// TwinCAT 3 PLC project PLC_TMO_VAC
// Title: PLC_TMO_VAC
// Company: SLAC - LCLS
// ProjectVersion: 0.0.0
// ProgramVersion: 3.1.4022.7
// CompilerDefines: K
// libraries:
//   LCLS General, * (SLAC)
//   LCLS Vacuum, * (SLAC - LCLS)
//   LCLSVacuumSerialDriverLib, * (SLAC - LCLS)
//   PMPS, * (SLAC - LCLS)
//   Tc2_SerialCom, * (Beckhoff Automation GmbH)
//   Tc2_Standard, * (Beckhoff Automation GmbH)
//   Tc2_System, * (Beckhoff Automation GmbH)
//   Tc3_Module, * (Beckhoff Automation GmbH)
// project tree:
//   / ComTask.TcTTO, FSVTask.TcTTO, PlcTask.TcTTO
//   DUTs/ E_STATES.TcDUT
//   GVLs/ GVL_COM.TcGVL, GVL_DREAM_ECAT.TcGVL, GVL_FEE_Device.TcGVL, GVL_FSV_PMPS.TcGVL, GVL_FS_Devices.TcGVL, GVL_Hutch_Gauges.TcGVL, GVL_Hutch_Pumps.TcGVL, GVL_Hutch_Valves.TcGVL, GVL_IP1_ECAT.TcGVL, GVL_PMPS.TcGVL, GVL_Variables.TcGVL
//   POUs/ DIAGNOSTICS.TcPOU, FB_VRC_NO_FFO_VLS.TcPOU, F_Turbo_Protection_ILK.TcPOU, MAIN.TcPOU, PRG_COM.TcPOU, PRG_FEE.TcPOU, PRG_FSV.TcPOU, PRG_FSV_Interfaces.TcPOU, PRG_Hutch_Beamline_Valves.TcPOU, PRG_Hutch_Gauges.TcPOU, PRG_Hutch_Ion_Pumps.TcPOU, PRG_HV_SAFETY.TcPOU, PRG_IP1_ECAT_Interfaces.TcPOU, PRG_PMPS.TcPOU, PRG_Roughing_Pumps.TcPOU, PRG_ECAT_COMM_CHECK.TcPOU
// real-time tasks:
//   TASK PlcTask: cycle T#10ms, priority 20, ADS port 350
//   TASK ComTask: cycle T#11ms, priority 30, ADS port 351
//   TASK FSVTask: cycle T#2ms, priority 15, ADS port 352
// I/O:
//   DEVICE Device 1 (EtherCAT), AmsNetId 172.21.132.78.2.1
//     B940-R20-CX0 (EK1200) [EK1200-5000 EtherCAT Power supply (2A E-Bus)]
//       CX0_E1 (EL2202) [EL2202 2Ch. Dig. Output 24V, 0.5A]
//       CX0_E1A (EL2202) [EL2202 2Ch. Dig. Output 24V, 0.5A]
//       Term 113 (EL2202) [EL2202 2Ch. Dig. Output 24V, 0.5A]
//       CX0_E2_EXILK (EL1008) [EL1008 8Ch. Dig. Input 24V, 3ms]
//       CX0_E5 (EL6070) [EL6070 1Ch. Licensing-Terminal]
//       CX0_E6_QPC1 (EL3064) [EL3064 4Ch. Ana. Input 0-10V]
//       CX0_E7_QPC1 (EL1004) [EL1004 4Ch. Dig. Input 24V, 3ms]
//       CX0_E8_QPC1 (EL2794) [EL2794 4Ch. Dig. Output 24V AC/DC, 2A, short-circuit-proof]
//       CX0_E9_QPC2 (EL3064) [EL3064 4Ch. Ana. Input 0-10V]
//       CX0_E10_QPC2 (EL1004) [EL1004 4Ch. Dig. Input 24V, 3ms]
//       CX0_E11_QPC2 (EL2794) [EL2794 4Ch. Dig. Output 24V AC/DC, 2A, short-circuit-proof]
//       CX0_E12 (EL6001) [EL6001 Interface (RS232)]
//       CX0_E13 (EK1122) [EK1122 2 port EtherCAT junction]
//         IP1_ECAT [EL6695 EtherCAT Bridge terminal (Secondary)]
//         DREAM_ECAT [EL6695 EtherCAT Bridge terminal (Secondary)]
//       PMPS_PRE [EL6692 EtherCAT Bridge terminal (Primary)]
//       CX0_EK1110 [EK1110 EtherCAT extension]
//     B940_R20_EK0 (EK1100) [EK1100 EtherCAT Coupler (2A E-Bus)]
//       R20_EK0_E1_MKS937B (EL3064)
//       R20_EK0_E2_MKS937B (EL3064) [EL3064 4Ch. Ana. Input 0-10V]
//       R20_EK0_E3_MKS937B (EL2794) [EL2794 4Ch. Dig. Output 24V AC/DC, 2A, short-circuit-proof]
//       R20_EK0_SIP (EL3174-0002) [EL3174-0002 4Ch. Ana. Input +/-10V, +/-20mA 16 Bit, Isolated Channels]
//       R20_EK0_E4_MKS937B (EL9505) [EL9505 Power supply terminal 5V]
//       R20_EK0_E5_MKS937B (EL1124)
//       R20_EK0_E5A_MKS937B (EL1124) [EL1124 4Ch. Dig. Input 5V, 10µs, Sensor Power]
//       R20_EK0_E6_MKS937B (EK1110) [EK1110 EtherCAT extension]
//     B940_K4S20_EK0  (EK1100) [EK1100 EtherCAT Coupler (2A E-Bus)]
//       K4S20-E1-FSV (EL1004)
//       K4S20-E2-FSV (EL2202) [EL2202 2Ch. Dig. Output 24V, 0.5A]
//       K4S20-E3-FSV (EL2202)
//       K4S20-E4-FSV (EK1110)
//     B940_K4S20_EB1  (EP2338-0002) [EP2338-0002 8 Ch. Dig. Input/Output 24V, 0,5A, M12]
//     B940_K4S20_EB2  (EP3174-0002) [EP3174-0002 4Ch. Ana. Input +/-10V, 0-10V, 0/4-20mA configurable]
//     B940_K4S20_EB3 (EP2624-0002) [EP2624-0002 4Ch. Relay Output, NO (125V AC / 30V DC)]
//     B940_K4S24_EB1 (EP3174-0002) [EP3174-0002 4Ch. Ana. Input +/-10V, 0-10V, 0/4-20mA configurable]
//     B940_K4S24_EB2 (EP2624-0002) [EP2624-0002 4Ch. Relay Output, NO (125V AC / 30V DC)]
//     B940_K4S28_EB1 (EP3174-0002) [EP3174-0002 4Ch. Ana. Input +/-10V, 0-10V, 0/4-20mA configurable]
//     B940_K4S28_EB2 (EP2624-0002) [EP2624-0002 4Ch. Relay Output, NO (125V AC / 30V DC)]
//     B940_K4S33_EB1 (EP2338-0002) [EP2338-0002 8 Ch. Dig. Input/Output 24V, 0,5A, M12]
//     B940_K4S33_EB2 (EP3174-0002) [EP3174-0002 4Ch. Ana. Input +/-10V, 0-10V, 0/4-20mA configurable]
//     B940_K4S33_EB3 (EP2624-0002) [EP2624-0002 4Ch. Relay Output, NO (125V AC / 30V DC)]
//     TMO_WALL_WEST_EP01 (EP4374-0002) [EP4374-0002 2Ch. Ana. Input +/-10V, 0-10V, 0/4-20mA configurable; 2Ch. Ana. Output +/-10V, 0-10V, 0/4-20mA configurable]
//     TMO_K4S2_DRL_01 (EK1100) [EK1100 EtherCAT Coupler (2A E-Bus)]
//       K4S2_01_E1_VFS (EL1004) [EL1004 4Ch. Dig. Input 24V, 3ms]
//       K4S2_01_E2 (EL9190) [EL9190 Power Supplier]
//       K4S2_01_E3_VFS (EL2202) [EL2202 2Ch. Dig. Output 24V, 0.5A]
//       K4S2_01_E4_VFS (EL2202) [EL2202 2Ch. Dig. Output 24V, 0.5A]
//       K4S2_01_E5 (EL1004)
//       K4S2_01_E6 (EL2004) [EL2004 4Ch. Dig. Output 24V, 0.5A]
//       Term 62 (EL9011) [EL9011 End Terminal]
//     TMO_K4S2_DRL_02 (EK1100) [EK1100 EtherCAT Coupler (2A E-Bus)]
//       K4S2_02_E1 (EL3174) [EL3174 4Ch. Ana. Input +/-10V Diff., +/-20mA SingleEnded, 16 Bit]
//       K4S2_02_E2 (EL3174) [EL3174 4Ch. Ana. Input +/-10V Diff., +/-20mA SingleEnded, 16 Bit]
//       K4S2_02_E3 (EL9184) [EL9184 Potential Connection, 8 x 24V, 8 x Ground]
//       K4S2_02_E4 (EL9070) [EL9070 Shield terminal]
//       K4S2_02_E5 (EL2624) [EL2624 4Ch. Relay Output, NO (125V AC / 30V DC)]
//       K4S2_02_E6 (EL9505) [EL9505 Power supply terminal 5V]
//       K4S2_02_E7 (EL1124) [EL1124 4Ch. Dig. Input 5V, 10µs, Sensor Power]
//       K4S2_02_E8 (EL1124) [EL1124 4Ch. Dig. Input 5V, 10µs, Sensor Power]
//       K4S2_02_E9 (EL9410) [EL9410 E-Bus Power Supplier  (Diagnostics)]
//       K4S2_02_E10 (EL6021) [EL6021 Interface (RS422/485)]
//       K4S2_02_E11 (EL1004) [EL1004 4Ch. Dig. Input 24V, 3ms]
//       K4S2_02_E12 (EL2794) [EL2794 4Ch. Dig. Output 24V AC/DC, 2A, short-circuit-proof]
//       K4S2_02_E13 (EL1004) [EL1004 4Ch. Dig. Input 24V, 3ms]
//       K4S2_02_E14 (EL2794) [EL2794 4Ch. Dig. Output 24V AC/DC, 2A, short-circuit-proof]
//       K4S2_02_E15 (EL1004) [EL1004 4Ch. Dig. Input 24V, 3ms]
//       K4S2_02_E16 (EL2794) [EL2794 4Ch. Dig. Output 24V AC/DC, 2A, short-circuit-proof]
//       K4S2_02_E17 (EL6001) [EL6001 Interface (RS232)]
//       K4S2_02_E18 (EL6001) [EL6001 Interface (RS232)]
//       K4S2_02_E19 (EL1004) [EL1004 4Ch. Dig. Input 24V, 3ms]
//       K4S2_02_E20 (EL2004) [EL2004 4Ch. Dig. Output 24V, 0.5A]
//       K4S2_02_E20A (EL1088) [EL1088 8Ch. Dig. Input 24V, 3ms, negative]
//       K4S2_02_E20 (EK1122) [EK1122 2 port EtherCAT junction]
//       Term 94 (EL9011) [EL9011 End Terminal]
//     TMO_K4S2_ EP1 (EP4374-0002) [EP4374-0002 2Ch. Ana. Input +/-10V, 0-10V, 0/4-20mA configurable; 2Ch. Ana. Output +/-10V, 0-10V, 0/4-20mA configurable]
//     TMO_K4S6_ EP1 (EP4374-0002) [EP4374-0002 2Ch. Ana. Input +/-10V, 0-10V, 0/4-20mA configurable; 2Ch. Ana. Output +/-10V, 0-10V, 0/4-20mA configurable]
//     TMO_K4S6_DRL_01 (EK1100) [EK1100 EtherCAT Coupler (2A E-Bus)]
//       K4S6_01_E1 (EL1004) [EL1004 4Ch. Dig. Input 24V, 3ms]
//       K4S6_01_E2 (EL2004) [EL2004 4Ch. Dig. Output 24V, 0.5A]
//       K4S6_01_E3 (EL1004) [EL1004 4Ch. Dig. Input 24V, 3ms]
//       K4S6_01_E4 (EL2004) [EL2004 4Ch. Dig. Output 24V, 0.5A]
//       K4S6_01_E5 (EL6021) [EL6021 Interface (RS422/485)]
//       K4S6_01_E6 (EL1004) [EL1004 4Ch. Dig. Input 24V, 3ms]
//       K4S6_01_E7 (EL2004) [EL2004 4Ch. Dig. Output 24V, 0.5A]
//       K4S6_01_E8 (EL1004) [EL1004 4Ch. Dig. Input 24V, 3ms]
//       K4S6_01_E9 (EL2004) [EL2004 4Ch. Dig. Output 24V, 0.5A]
//       K4S6_01_E10 (EL6021) [EL6021 Interface (RS422/485)]
//       K4S6_01_E11 (EL1004) [EL1004 4Ch. Dig. Input 24V, 3ms]
//       K4S6_01_E12 (EL2004) [EL2004 4Ch. Dig. Output 24V, 0.5A]
//       K4S6_01_E13 (EL9410) [EL9410 E-Bus Power Supplier  (Diagnostics)]
//       K4S6_01_E14 (EL2624) [EL2624 4Ch. Relay Output, NO (125V AC / 30V DC)]
//       K4S6_01_E15 (EL3174) [EL3174 4Ch. Ana. Input +/-10V Diff., +/-20mA SingleEnded, 16 Bit]
//       K4S6_01_E16 (EL9184) [EL9184 Potential Connection, 8 x 24V, 8 x Ground]
//       K4S6_01_E17 (EL9070) [EL9070 Shield terminal]
//       K4S6_01_E18 (EL3174) [EL3174 4Ch. Ana. Input +/-10V Diff., +/-20mA SingleEnded, 16 Bit]
//       K4S6_01_E19 (EL9505) [EL9505 Power supply terminal 5V]
//       K4S6_01_E20 (EL1124) [EL1124 4Ch. Dig. Input 5V, 10µs, Sensor Power]
//       K4S6_01_E21 (EL1124) [EL1124 4Ch. Dig. Input 5V, 10µs, Sensor Power]
//       Term 119 (EL9410) [EL9410 E-Bus Power Supplier  (Diagnostics)]
//       K4S6_01_E22_IP1 (EL1004) [EL1004 4Ch. Dig. Input 24V, 3ms]
//       K4S6_01_E23_IP1 (EL2794) [EL2794 4Ch. Dig. Output 24V AC/DC, 2A, short-circuit-proof]
//       Term 91 (EL9011) [EL9011 End Terminal]
//     TMO_K4S8_DRL_01 (EK1100) [EK1100 EtherCAT Coupler (2A E-Bus)]
//       K4S8_01_E1 (EL1004) [EL1004 4Ch. Dig. Input 24V, 3ms]
//       K4S8_01_E2 (EL9190) [EL9190 Power Supplier]
//       K4S8_01_E3 (EL2202) [EL2202 2Ch. Dig. Output 24V, 0.5A]
//       K4S8_01_E4 (EL2202) [EL2202 2Ch. Dig. Output 24V, 0.5A]
//       K4S8_01_E5 (EL1004) [EL1004 4Ch. Dig. Input 24V, 3ms]
//       K4S8_01_E6 (EL2004) [EL2004 4Ch. Dig. Output 24V, 0.5A]
//       K4S8_01_E6 (EK1122) [EK1122 2 port EtherCAT junction]
//       Term 92 (EL9011) [EL9011 End Terminal]
//     TMO_K4S8_DRL_02 (EK1100) [EK1100 EtherCAT Coupler (2A E-Bus)]
//       K4S8_02_E1 (EL1004) [EL1004 4Ch. Dig. Input 24V, 3ms]
//       K4S8_02_E2 (EL2004) [EL2004 4Ch. Dig. Output 24V, 0.5A]
//       K4S8_02_E3 (EL2624) [EL2624 4Ch. Relay Output, NO (125V AC / 30V DC)]
//       K4S8_02_E4 (EL3174) [EL3174 4Ch. Ana. Input +/-10V Diff., +/-20mA SingleEnded, 16 Bit]
//       K4S8_02_E5 (EL9184) [EL9184 Potential Connection, 8 x 24V, 8 x Ground]
//       K4S8_02_E6 (EL9070) [EL9070 Shield terminal]
//       K4S8_02_E6A (EL1084) [EL1084 4Ch. Dig. Input 24V, 3ms, negative]
//       K4S8_02_E7 (EL9505) [EL9505 Power supply terminal 5V]
//       K4S8_02_E8 (EL1124) [EL1124 4Ch. Dig. Input 5V, 10µs, Sensor Power]
//       END (EL9011) [EL9011 End Terminal]
// variable links:
//   PLC_TMO_VAC Instance <-> Device 1 (EtherCAT)/B940-R20-CX0 (EK1200)/CX0_E1 (EL2202)
//     PlcTask Outputs/GVL_PMPS.g_FastFaultOutput1.q_xFastFaultOut <-> Channel 1/Output
//     PlcTask Outputs/GVL_PMPS.g_FastFaultOutput2.q_xFastFaultOut <-> Channel 2/Output
//   PLC_TMO_VAC Instance <-> Device 1 (EtherCAT)/B940-R20-CX0 (EK1200)/CX0_E10_QPC2 (EL1004)
//     PlcTask Inputs/GVL_FEE_Device.PC4K4_XTES_PIP_01.i_xSP_DI <-> Channel 1/Input
//     PlcTask Inputs/GVL_FEE_Device.TV1K4_PIP_01.i_xSP_DI <-> Channel 3/Input
//     PlcTask Inputs/GVL_Hutch_Pumps.MR2K4_KBO_PIP_01.i_xSP_DI <-> Channel 2/Input
//     PlcTask Inputs/GVL_Hutch_Pumps.MR4K4_KBO_PIP_01.i_xSP_DI <-> Channel 4/Input
//   PLC_TMO_VAC Instance <-> Device 1 (EtherCAT)/B940-R20-CX0 (EK1200)/CX0_E11_QPC2 (EL2794)
//     PlcTask Outputs/GVL_FEE_Device.PC4K4_XTES_PIP_01.q_xHVEna_DO <-> Channel 1/Output
//     PlcTask Outputs/GVL_FEE_Device.TV1K4_PIP_01.q_xHVEna_DO <-> Channel 3/Output
//     PlcTask Outputs/GVL_Hutch_Pumps.MR2K4_KBO_PIP_01.q_xHVEna_DO <-> Channel 2/Output
//     PlcTask Outputs/GVL_Hutch_Pumps.MR4K4_KBO_PIP_01.q_xHVEna_DO <-> Channel 4/Output
//   PLC_TMO_VAC Instance <-> Device 1 (EtherCAT)/B940-R20-CX0 (EK1200)/CX0_E13 (EK1122)/DREAM_ECAT (EL6695-0002)
//     ComTask Inputs/GVL_DREAM_ECAT.DREAM_HV_SAFETY_ENABLE <-> IO Inputs/DREAM_HV_SAFETY_ENABLE
//     ComTask Inputs/GVL_DREAM_ECAT.DREAM_PLC_NAME <-> IO Inputs/ENDSTATION_PLC_NAME
//     ComTask Inputs/GVL_DREAM_ECAT.DREAM_TURBOS_ALL_AtSpd <-> IO Inputs/DREAM_TURBOS_ALL_AtSpd
//     ComTask Outputs/GVL_DREAM_ECAT.sHutchPlcName <-> IO Outputs/HUTCH_PLC_NAME
//     PlcTask Inputs/GVL_DREAM_ECAT.DREAM_MAIN_GAUGE.i_rPRESS <-> IO Inputs/DREAM_MAIN_rPRESS
//     PlcTask Inputs/GVL_DREAM_ECAT.DREAM_MAIN_GAUGE.i_xAT_VAC <-> IO Inputs/DREAM_MAIN_xAT_VAC
//     PlcTask Inputs/GVL_DREAM_ECAT.DREAM_MAIN_GAUGE.i_xPRESS_OK <-> IO Inputs/DREAM_MAIN_xPRESS_OK
//     PlcTask Inputs/GVL_DREAM_ECAT.bDreamEcatBridge_External_device_not_connected <-> SYNC Inputs/External device not connected
//     PlcTask Inputs/GVL_DREAM_ECAT.bDreamEcatBridge_TxPDO_state <-> SYNC Inputs/TxPDO state
//     PlcTask Inputs/GVL_DREAM_ECAT.bDreamEcatBridge_WcState <-> WcState/WcState
//   PLC_TMO_VAC Instance <-> Device 1 (EtherCAT)/B940-R20-CX0 (EK1200)/CX0_E13 (EK1122)/IP1_ECAT (EL6692)
//     ComTask Inputs/GVL_IP1_ECAT.IP1_HV_SAFETY_ENABLE <-> IO Inputs/IP1_HV_SAFETY_ENABLE
//     ComTask Inputs/GVL_IP1_ECAT.IP1_PLC_NAME <-> IO Inputs/ENDSTATION_PLC_NAME
//     ComTask Outputs/GVL_IP1_ECAT.My_PLC_NAME <-> IO Outputs/HUTCH_PLC_NAME
//     PlcTask Inputs/GVL_IP1_ECAT.IP1_MAIN_GAUGE.i_rPRESS <-> IO Inputs/IP1_MAIN_rPRESS
//     PlcTask Inputs/GVL_IP1_ECAT.IP1_MAIN_GAUGE.i_xAT_VAC <-> IO Inputs/IP1_MAIN_xAT_VAC
//     PlcTask Inputs/GVL_IP1_ECAT.IP1_MAIN_GAUGE.i_xPRESS_OK <-> IO Inputs/IP1_MAIN_xPRESS_OK
//     PlcTask Inputs/GVL_IP1_ECAT.IP1_ROUGH_VRC_01_AtOpnLS <-> IO Inputs/IP1_ROUGH_VRC_01_OPEN_LS
//     PlcTask Inputs/GVL_IP1_ECAT.IP1_ROUGH_VRC_02_AtOpnLS <-> IO Inputs/IP1_ROUGH_VRC_02_OPEN_LS
//     PlcTask Inputs/GVL_IP1_ECAT.IP1_ROUGH_VRC_03_AtOpnLS <-> IO Inputs/IP1_ROUGH_VRC_03_OPEN_LS
//     PlcTask Inputs/GVL_IP1_ECAT.IP1_TURBOS_ALL_AtSpd <-> IO Inputs/IP1_TURBOS_ALL_AtSpd
//     PlcTask Inputs/GVL_IP1_ECAT.xEcatBridge_External_device_not_connected <-> SYNC Inputs/External device not connected
//     PlcTask Inputs/GVL_IP1_ECAT.xEcatBridge_TxPDO_state <-> SYNC Inputs/TxPDO state
//     PlcTask Inputs/GVL_IP1_ECAT.xEcatBridge_WcState <-> WcState/WcState
//     PlcTask Outputs/GVL_IP1_ECAT.ROUGH1_VRC_01_AtOpnLS <-> IO Outputs/TMO_ROUGH1_VRC_01_OPEN_LS
//     PlcTask Outputs/GVL_IP1_ECAT.ROUGH2_VRC_01_AtOpnLS <-> IO Outputs/TMO_ROUGH2_VRC_01_OPEN_LS
//   PLC_TMO_VAC Instance <-> Device 1 (EtherCAT)/B940-R20-CX0 (EK1200)/CX0_E1A (EL2202)
//     FSVTask Outputs/GVL_PMPS.g_FastFaultOutput3.q_xFastFaultOut <-> Channel 1/Output
//     FSVTask Outputs/GVL_PMPS.g_FastFaultOutput4.q_xFastFaultOut <-> Channel 2/Output
//   PLC_TMO_VAC Instance <-> Device 1 (EtherCAT)/B940-R20-CX0 (EK1200)/CX0_E2_EXILK (EL1008)
//     PlcTask Inputs/GVL_FEE_Device.USVacOk_HI <-> Channel 1/Input
//     PlcTask Inputs/GVL_FEE_Device.USVacOk_LO <-> Channel 3/Input
//   PLC_TMO_VAC Instance <-> Device 1 (EtherCAT)/B940-R20-CX0 (EK1200)/CX0_E6_QPC1 (EL3064)
//     PlcTask Inputs/GVL_FEE_Device.MR1K4_SOMS_PIP_01.i_iPRESS <-> AI Standard Channel 1/Value
//     PlcTask Inputs/GVL_FEE_Device.ST1K4_TEST_PIP_01.i_iPRESS <-> AI Standard Channel 2/Value
//     PlcTask Inputs/GVL_FEE_Device.ST2K4_BCS_PIP_01.i_iPRESS <-> AI Standard Channel 3/Value
//     PlcTask Inputs/GVL_FEE_Device.ST3K4_PPS_PIP_01.i_iPRESS <-> AI Standard Channel 4/Value
//   PLC_TMO_VAC Instance <-> Device 1 (EtherCAT)/B940-R20-CX0 (EK1200)/CX0_E7_QPC1 (EL1004)
//     PlcTask Inputs/GVL_FEE_Device.MR1K4_SOMS_PIP_01.i_xSP_DI <-> Channel 1/Input
//     PlcTask Inputs/GVL_FEE_Device.ST1K4_TEST_PIP_01.i_xSP_DI <-> Channel 2/Input
//     PlcTask Inputs/GVL_FEE_Device.ST2K4_BCS_PIP_01.i_xSP_DI <-> Channel 3/Input
//     PlcTask Inputs/GVL_FEE_Device.ST3K4_PPS_PIP_01.i_xSP_DI <-> Channel 4/Input
//   PLC_TMO_VAC Instance <-> Device 1 (EtherCAT)/B940-R20-CX0 (EK1200)/CX0_E8_QPC1 (EL2794)
//     PlcTask Outputs/GVL_FEE_Device.MR1K4_SOMS_PIP_01.q_xHVEna_DO <-> Channel 1/Output
//     PlcTask Outputs/GVL_FEE_Device.ST1K4_TEST_PIP_01.q_xHVEna_DO <-> Channel 2/Output
//     PlcTask Outputs/GVL_FEE_Device.ST2K4_BCS_PIP_01.q_xHVEna_DO <-> Channel 3/Output
//     PlcTask Outputs/GVL_FEE_Device.ST3K4_PPS_PIP_01.q_xHVEna_DO <-> Channel 4/Output
//   PLC_TMO_VAC Instance <-> Device 1 (EtherCAT)/B940-R20-CX0 (EK1200)/CX0_E9_QPC2 (EL3064)
//     PlcTask Inputs/GVL_FEE_Device.PC4K4_XTES_PIP_01.i_iPRESS <-> AI Standard Channel 1/Value
//     PlcTask Inputs/GVL_FEE_Device.TV1K4_PIP_01.i_iPRESS <-> AI Standard Channel 3/Value
//     PlcTask Inputs/GVL_Hutch_Pumps.MR2K4_KBO_PIP_01.i_iPRESS <-> AI Standard Channel 2/Value
//     PlcTask Inputs/GVL_Hutch_Pumps.MR4K4_KBO_PIP_01.i_iPRESS <-> AI Standard Channel 4/Value
//   PLC_TMO_VAC Instance <-> Device 1 (EtherCAT)/B940-R20-CX0 (EK1200)/PMPS_PRE
//     PlcTask Inputs/PRG_PMPS.fbArbiterIO.i_stCurrentBP <-> IO Inputs/CurrentBP
//     PlcTask Inputs/PRG_PMPS.fbArbiterIO.xTxPDO_state <-> SYNC Inputs/TxPDO state
//     PlcTask Inputs/PRG_PMPS.fbArbiterIO.xTxPDO_toggle <-> SYNC Inputs/TxPDO toggle
//     PlcTask Outputs/PRG_PMPS.fbArbiterIO.q_stRequestedBP <-> IO Outputs/RequestedBP
//   PLC_TMO_VAC Instance <-> Device 1 (EtherCAT)/B940_K4S20_EB1  (EP2338-0002)
//     PlcTask Inputs/GVL_FEE_Device.TV1K4_VGC_01.i_xClsLS <-> Channel 2/Input
//     PlcTask Inputs/GVL_FEE_Device.TV1K4_VGC_02.i_xClsLS <-> Channel 6/Input
//     PlcTask Inputs/GVL_FEE_Device.TV1K4_VGC_01.i_xOpnLS <-> Channel 1/Input
//     PlcTask Inputs/GVL_FEE_Device.TV1K4_VGC_02.i_xOpnLS <-> Channel 5/Input
//     PlcTask Outputs/GVL_FEE_Device.TV1K4_VGC_01.q_xOPN_DO <-> Channel 11/Output
//     PlcTask Outputs/GVL_FEE_Device.TV1K4_VGC_02.q_xOPN_DO <-> Channel 15/Output
//   PLC_TMO_VAC Instance <-> Device 1 (EtherCAT)/B940_K4S20_EB2  (EP3174-0002)
//     PlcTask Inputs/GVL_FEE_Device.TV1K4_GCC_01.i_iPRESS_R <-> AI Standard Channel 2/Value
//     PlcTask Inputs/GVL_FEE_Device.TV1K4_GPI_01.i_iPRESS_R <-> AI Standard Channel 1/Value
//   PLC_TMO_VAC Instance <-> Device 1 (EtherCAT)/B940_K4S20_EB3 (EP2624-0002)
//     PlcTask Outputs/GVL_FEE_Device.TV1K4_GCC_01.q_xHV_DIS <-> Channel 1/Output
//   PLC_TMO_VAC Instance <-> Device 1 (EtherCAT)/B940_K4S20_EK0  (EK1100)/K4S20-E1-FSV (EL1004)
//     FSVTask Inputs/GVL_FS_Devices.TV1K4_VFS_1.i_xClsLS <-> Channel 1/Input
//     FSVTask Inputs/GVL_FS_Devices.TV1K4_VFS_1.i_xOpnLS <-> Channel 2/Input
//   PLC_TMO_VAC Instance <-> Device 1 (EtherCAT)/B940_K4S20_EK0  (EK1100)/K4S20-E2-FSV (EL2202)
//     FSVTask Outputs/GVL_FS_Devices.TV1K4_VFS_1.q_xClose_A <-> Channel 1/Output
//     FSVTask Outputs/GVL_FS_Devices.TV1K4_VFS_1.q_xClose_B <-> Channel 2/Output
//   PLC_TMO_VAC Instance <-> Device 1 (EtherCAT)/B940_K4S20_EK0  (EK1100)/K4S20-E3-FSV (EL2202)
//     FSVTask Outputs/GVL_FS_Devices.TV1K4_VFS_1.q_xClose_C <-> Channel 1/Output
//     FSVTask Outputs/GVL_FS_Devices.TV1K4_VFS_1.q_xOPN_DO <-> Channel 2/Output
//   PLC_TMO_VAC Instance <-> Device 1 (EtherCAT)/B940_K4S24_EB1 (EP3174-0002)
//     PlcTask Inputs/GVL_FEE_Device.ST1K4_TEST_GCC_01.i_iPRESS_R <-> AI Standard Channel 2/Value
//     PlcTask Inputs/GVL_FEE_Device.ST1K4_TEST_GPI_01.i_iPRESS_R <-> AI Standard Channel 1/Value
//   PLC_TMO_VAC Instance <-> Device 1 (EtherCAT)/B940_K4S24_EB2 (EP2624-0002)
//     PlcTask Outputs/GVL_FEE_Device.ST1K4_TEST_GCC_01.q_xHV_DIS <-> Channel 1/Output
//   PLC_TMO_VAC Instance <-> Device 1 (EtherCAT)/B940_K4S28_EB1 (EP3174-0002)
//     PlcTask Inputs/GVL_FEE_Device.ST2K4_BCS_GCC_01.i_iPRESS_R <-> AI Standard Channel 2/Value
//     PlcTask Inputs/GVL_FEE_Device.ST2K4_BCS_GPI_01.i_iPRESS_R <-> AI Standard Channel 1/Value
//   PLC_TMO_VAC Instance <-> Device 1 (EtherCAT)/B940_K4S28_EB2 (EP2624-0002)
//     PlcTask Outputs/GVL_FEE_Device.ST2K4_BCS_GCC_01.q_xHV_DIS <-> Channel 1/Output
//   PLC_TMO_VAC Instance <-> Device 1 (EtherCAT)/B940_K4S33_EB1 (EP2338-0002)
//     PlcTask Inputs/GVL_FEE_Device.ST3K4_PPS_VGC_01.i_xClsLS <-> Channel 2/Input
//     PlcTask Inputs/GVL_FEE_Device.ST3K4_PPS_VGC_01.i_xOpnLS <-> Channel 1/Input
//     PlcTask Outputs/GVL_FEE_Device.ST3K4_PPS_VGC_01.q_xOPN_DO <-> Channel 11/Output
//   PLC_TMO_VAC Instance <-> Device 1 (EtherCAT)/B940_K4S33_EB2 (EP3174-0002)
//     PlcTask Inputs/GVL_FEE_Device.PC4K4_XTES_GCC_01.i_iPRESS_R <-> AI Standard Channel 2/Value
//     PlcTask Inputs/GVL_FEE_Device.PC4K4_XTES_GPI_01.i_iPRESS_R <-> AI Standard Channel 1/Value
//   PLC_TMO_VAC Instance <-> Device 1 (EtherCAT)/B940_K4S33_EB3 (EP2624-0002)
//     PlcTask Outputs/GVL_FEE_Device.PC4K4_XTES_GCC_01.q_xHV_DIS <-> Channel 1/Output
//   PLC_TMO_VAC Instance <-> Device 1 (EtherCAT)/B940_R20_EK0 (EK1100)/R20_EK0_E1_MKS937B (EL3064)
//     PlcTask Inputs/GVL_Hutch_Gauges.LI2K4_IP1_GFS_01.i_iPRESS_R <-> AI Standard Channel 1/Value
//     PlcTask Inputs/GVL_Hutch_Gauges.LI2K4_IP1_GFS_02.i_iPRESS_R <-> AI Standard Channel 2/Value
//   PLC_TMO_VAC Instance <-> Device 1 (EtherCAT)/B940_R20_EK0 (EK1100)/R20_EK0_E2_MKS937B (EL3064)
//     PlcTask Inputs/GVL_Hutch_Gauges.LI2K4_IP1_GFS_03.i_iPRESS_R <-> AI Standard Channel 1/Value
//   PLC_TMO_VAC Instance <-> Device 1 (EtherCAT)/B940_R20_EK0 (EK1100)/R20_EK0_E3_MKS937B (EL2794)
//     PlcTask Outputs/GVL_Hutch_Gauges.LI2K4_IP1_GFS_01.q_xHV_DIS <-> Channel 1/Output
//     PlcTask Outputs/GVL_Hutch_Gauges.LI2K4_IP1_GFS_02.q_xHV_DIS <-> Channel 2/Output
//     PlcTask Outputs/GVL_Hutch_Gauges.LI2K4_IP1_GFS_03.q_xHV_DIS <-> Channel 3/Output
//     PlcTask Outputs/GVL_Hutch_Pumps.PA2K4_IP1_PIP_01.q_xHVEna_DO <-> Channel 4/Output
//   PLC_TMO_VAC Instance <-> Device 1 (EtherCAT)/B940_R20_EK0 (EK1100)/R20_EK0_E5A_MKS937B (EL1124)
//     FSVTask Inputs/GVL_FS_Devices.MR3K4_KBO_VFS_1.i_xTriggerIG3 <-> Channel 1/Input
//     FSVTask Inputs/GVL_FS_Devices.MR4K4_KBO_VFS_1.i_xTriggerIG3 <-> Channel 1/Input
//     FSVTask Inputs/GVL_FS_Devices.TV1K4_VFS_1.i_xTriggerIG3 <-> Channel 1/Input
//   PLC_TMO_VAC Instance <-> Device 1 (EtherCAT)/B940_R20_EK0 (EK1100)/R20_EK0_E5_MKS937B (EL1124)
//     FSVTask Inputs/GVL_FS_Devices.MR3K4_KBO_VFS_1.i_xTriggerIG1 <-> Channel 1/Input
//     FSVTask Inputs/GVL_FS_Devices.MR3K4_KBO_VFS_1.i_xTriggerIG2 <-> Channel 2/Input
//     FSVTask Inputs/GVL_FS_Devices.MR4K4_KBO_VFS_1.i_xTriggerIG1 <-> Channel 1/Input
//     FSVTask Inputs/GVL_FS_Devices.MR4K4_KBO_VFS_1.i_xTriggerIG2 <-> Channel 2/Input
//     FSVTask Inputs/GVL_FS_Devices.TV1K4_VFS_1.i_xTriggerIG1 <-> Channel 1/Input
//     FSVTask Inputs/GVL_FS_Devices.TV1K4_VFS_1.i_xTriggerIG2 <-> Channel 2/Input
//     PlcTask Inputs/GVL_Hutch_Pumps.PA2K4_IP1_PIP_01.i_xError <-> Channel 4/Input
//     PlcTask Inputs/GVL_Hutch_Pumps.PA2K4_IP1_PIP_01.i_xIP_ON <-> Channel 3/Input
//   PLC_TMO_VAC Instance <-> Device 1 (EtherCAT)/B940_R20_EK0 (EK1100)/R20_EK0_SIP (EL3174-0002)
//     PlcTask Inputs/GVL_Hutch_Pumps.PA2K4_IP1_PIP_01.i_iPRESS <-> AI Standard Channel 1/Value
//   PLC_TMO_VAC Instance <-> Device 1 (EtherCAT)/TMO_K4S2_ EP1 (EP4374-0002)
//     PlcTask Inputs/GVL_Hutch_Gauges.TMO_ROUGH1_GPI_02.i_iPRESS_R <-> AI Inputs Channel 1/Value
//     PlcTask Inputs/GVL_Hutch_Gauges.TMO_ROUGH2_GPI_02.i_iPRESS_R <-> AI Inputs Channel 2/Value
//     PlcTask Outputs/GVL_Hutch_Valves.TMO_ROUGH1_VFV_02.q_iRawPosition <-> AO Outputs Channel 3/Analog output
//     PlcTask Outputs/GVL_Hutch_Valves.TMO_ROUGH2_VFV_01.q_iRawPosition <-> AO Outputs Channel 4/Analog output
//   PLC_TMO_VAC Instance <-> Device 1 (EtherCAT)/TMO_K4S2_DRL_01 (EK1100)/K4S2_01_E1_VFS (EL1004)
//     FSVTask Inputs/GVL_FS_Devices.MR3K4_KBO_VFS_1.i_xClsLS <-> Channel 1/Input
//     FSVTask Inputs/GVL_FS_Devices.MR3K4_KBO_VFS_1.i_xOpnLS <-> Channel 2/Input
//   PLC_TMO_VAC Instance <-> Device 1 (EtherCAT)/TMO_K4S2_DRL_01 (EK1100)/K4S2_01_E3_VFS (EL2202)
//     FSVTask Outputs/GVL_FS_Devices.MR3K4_KBO_VFS_1.q_xClose_A <-> Channel 1/Output
//     FSVTask Outputs/GVL_FS_Devices.MR3K4_KBO_VFS_1.q_xClose_B <-> Channel 2/Output
//   PLC_TMO_VAC Instance <-> Device 1 (EtherCAT)/TMO_K4S2_DRL_01 (EK1100)/K4S2_01_E4_VFS (EL2202)
//     FSVTask Outputs/GVL_FS_Devices.MR3K4_KBO_VFS_1.q_xClose_C <-> Channel 1/Output
//     FSVTask Outputs/GVL_FS_Devices.MR3K4_KBO_VFS_1.q_xOPN_DO <-> Channel 2/Output
//   PLC_TMO_VAC Instance <-> Device 1 (EtherCAT)/TMO_K4S2_DRL_01 (EK1100)/K4S2_01_E5 (EL1004)
//     PlcTask Inputs/GVL_Hutch_Valves.MR2K4_KBO_VWC_01.i_xClsLS <-> Channel 2/Input
//     PlcTask Inputs/GVL_Hutch_Valves.MR3K4_KBO_VWC_01.i_xClsLS <-> Channel 4/Input
//     PlcTask Inputs/GVL_Hutch_Valves.MR2K4_KBO_VWC_01.i_xOpnLS <-> Channel 1/Input
//     PlcTask Inputs/GVL_Hutch_Valves.MR3K4_KBO_VWC_01.i_xOpnLS <-> Channel 3/Input
//   PLC_TMO_VAC Instance <-> Device 1 (EtherCAT)/TMO_K4S2_DRL_01 (EK1100)/K4S2_01_E6 (EL2004)
//     PlcTask Outputs/GVL_Hutch_Valves.MR2K4_KBO_VWC_01.q_xOPN_DO <-> Channel 1/Output
//     PlcTask Outputs/GVL_Hutch_Valves.MR3K4_KBO_VWC_01.q_xOPN_DO <-> Channel 2/Output
//   PLC_TMO_VAC Instance <-> Device 1 (EtherCAT)/TMO_K4S2_DRL_02 (EK1100)/K4S2_02_E1 (EL3174)
//     PlcTask Inputs/GVL_Hutch_Gauges.MR2K4_KBO_GCC_01.i_iPRESS_R <-> AI Standard Channel 3/Value
//     PlcTask Inputs/GVL_Hutch_Gauges.MR2K4_KBO_GPI_01.i_iPRESS_R <-> AI Standard Channel 2/Value
//     PlcTask Inputs/GVL_Hutch_Gauges.PA1K4_IP1_GCC_01.i_iPRESS_R <-> AI Standard Channel 4/Value
//   PLC_TMO_VAC Instance <-> Device 1 (EtherCAT)/TMO_K4S2_DRL_02 (EK1100)/K4S2_02_E10 (EL6021)
//     ComTask Inputs/GVL_COM.K4S2_02_E10_stComIn/D[0] <-> COM TxPDO-Map Inputs/Data In 0
//     ComTask Inputs/GVL_COM.K4S2_02_E10_stComIn/D[10] <-> COM TxPDO-Map Inputs/Data In 10
//     ComTask Inputs/GVL_COM.K4S2_02_E10_stComIn/D[11] <-> COM TxPDO-Map Inputs/Data In 11
//     ComTask Inputs/GVL_COM.K4S2_02_E10_stComIn/D[12] <-> COM TxPDO-Map Inputs/Data In 12
//     ComTask Inputs/GVL_COM.K4S2_02_E10_stComIn/D[13] <-> COM TxPDO-Map Inputs/Data In 13
//     ComTask Inputs/GVL_COM.K4S2_02_E10_stComIn/D[14] <-> COM TxPDO-Map Inputs/Data In 14
//     ComTask Inputs/GVL_COM.K4S2_02_E10_stComIn/D[15] <-> COM TxPDO-Map Inputs/Data In 15
//     ComTask Inputs/GVL_COM.K4S2_02_E10_stComIn/D[16] <-> COM TxPDO-Map Inputs/Data In 16
//     ComTask Inputs/GVL_COM.K4S2_02_E10_stComIn/D[17] <-> COM TxPDO-Map Inputs/Data In 17
//     ComTask Inputs/GVL_COM.K4S2_02_E10_stComIn/D[18] <-> COM TxPDO-Map Inputs/Data In 18
//     ComTask Inputs/GVL_COM.K4S2_02_E10_stComIn/D[19] <-> COM TxPDO-Map Inputs/Data In 19
//     ComTask Inputs/GVL_COM.K4S2_02_E10_stComIn/D[1] <-> COM TxPDO-Map Inputs/Data In 1
//     ComTask Inputs/GVL_COM.K4S2_02_E10_stComIn/D[20] <-> COM TxPDO-Map Inputs/Data In 20
//     ComTask Inputs/GVL_COM.K4S2_02_E10_stComIn/D[21] <-> COM TxPDO-Map Inputs/Data In 21
//     ComTask Inputs/GVL_COM.K4S2_02_E10_stComIn/D[2] <-> COM TxPDO-Map Inputs/Data In 2
//     ComTask Inputs/GVL_COM.K4S2_02_E10_stComIn/D[3] <-> COM TxPDO-Map Inputs/Data In 3
//     ComTask Inputs/GVL_COM.K4S2_02_E10_stComIn/D[4] <-> COM TxPDO-Map Inputs/Data In 4
//     ComTask Inputs/GVL_COM.K4S2_02_E10_stComIn/D[5] <-> COM TxPDO-Map Inputs/Data In 5
//     ComTask Inputs/GVL_COM.K4S2_02_E10_stComIn/D[6] <-> COM TxPDO-Map Inputs/Data In 6
//     ComTask Inputs/GVL_COM.K4S2_02_E10_stComIn/D[7] <-> COM TxPDO-Map Inputs/Data In 7
//     ComTask Inputs/GVL_COM.K4S2_02_E10_stComIn/D[8] <-> COM TxPDO-Map Inputs/Data In 8
//     ComTask Inputs/GVL_COM.K4S2_02_E10_stComIn/D[9] <-> COM TxPDO-Map Inputs/Data In 9
//     ComTask Inputs/GVL_COM.K4S2_02_E10_stComIn/Status <-> COM TxPDO-Map Inputs/Status
//     ComTask Outputs/GVL_COM.K4S2_02_E10_stComOut/Ctrl <-> COM RxPDO-Map Outputs/Ctrl
//     ComTask Outputs/GVL_COM.K4S2_02_E10_stComOut/D[0] <-> COM RxPDO-Map Outputs/Data Out 0
//     ComTask Outputs/GVL_COM.K4S2_02_E10_stComOut/D[10] <-> COM RxPDO-Map Outputs/Data Out 10
//     ComTask Outputs/GVL_COM.K4S2_02_E10_stComOut/D[11] <-> COM RxPDO-Map Outputs/Data Out 11
//     ComTask Outputs/GVL_COM.K4S2_02_E10_stComOut/D[12] <-> COM RxPDO-Map Outputs/Data Out 12
//     ComTask Outputs/GVL_COM.K4S2_02_E10_stComOut/D[13] <-> COM RxPDO-Map Outputs/Data Out 13
//     ComTask Outputs/GVL_COM.K4S2_02_E10_stComOut/D[14] <-> COM RxPDO-Map Outputs/Data Out 14
//     ComTask Outputs/GVL_COM.K4S2_02_E10_stComOut/D[15] <-> COM RxPDO-Map Outputs/Data Out 15
//     ComTask Outputs/GVL_COM.K4S2_02_E10_stComOut/D[16] <-> COM RxPDO-Map Outputs/Data Out 16
//     ComTask Outputs/GVL_COM.K4S2_02_E10_stComOut/D[17] <-> COM RxPDO-Map Outputs/Data Out 17
//     ComTask Outputs/GVL_COM.K4S2_02_E10_stComOut/D[18] <-> COM RxPDO-Map Outputs/Data Out 18
//     ComTask Outputs/GVL_COM.K4S2_02_E10_stComOut/D[19] <-> COM RxPDO-Map Outputs/Data Out 19
//     ComTask Outputs/GVL_COM.K4S2_02_E10_stComOut/D[1] <-> COM RxPDO-Map Outputs/Data Out 1
//     ComTask Outputs/GVL_COM.K4S2_02_E10_stComOut/D[20] <-> COM RxPDO-Map Outputs/Data Out 20
//     ComTask Outputs/GVL_COM.K4S2_02_E10_stComOut/D[21] <-> COM RxPDO-Map Outputs/Data Out 21
//     ComTask Outputs/GVL_COM.K4S2_02_E10_stComOut/D[2] <-> COM RxPDO-Map Outputs/Data Out 2
//     ComTask Outputs/GVL_COM.K4S2_02_E10_stComOut/D[3] <-> COM RxPDO-Map Outputs/Data Out 3
//     ComTask Outputs/GVL_COM.K4S2_02_E10_stComOut/D[4] <-> COM RxPDO-Map Outputs/Data Out 4
//     ComTask Outputs/GVL_COM.K4S2_02_E10_stComOut/D[5] <-> COM RxPDO-Map Outputs/Data Out 5
//     ComTask Outputs/GVL_COM.K4S2_02_E10_stComOut/D[6] <-> COM RxPDO-Map Outputs/Data Out 6
//     ComTask Outputs/GVL_COM.K4S2_02_E10_stComOut/D[7] <-> COM RxPDO-Map Outputs/Data Out 7
//     ComTask Outputs/GVL_COM.K4S2_02_E10_stComOut/D[8] <-> COM RxPDO-Map Outputs/Data Out 8
//     ComTask Outputs/GVL_COM.K4S2_02_E10_stComOut/D[9] <-> COM RxPDO-Map Outputs/Data Out 9
//   PLC_TMO_VAC Instance <-> Device 1 (EtherCAT)/TMO_K4S2_DRL_02 (EK1100)/K4S2_02_E11 (EL1004)
//     PlcTask Inputs/GVL_Hutch_Pumps.PA1K4_IP1_PTM_01.i_xAtSpd <-> Channel 2/Input
//     PlcTask Inputs/GVL_Hutch_Pumps.PA1K4_IP1_PTM_02.i_xAtSpd <-> Channel 4/Input
//     PlcTask Inputs/GVL_Hutch_Pumps.PA1K4_IP1_PTM_01.i_xFaultNC <-> Channel 1/Input
//     PlcTask Inputs/GVL_Hutch_Pumps.PA1K4_IP1_PTM_02.i_xFaultNC <-> Channel 3/Input
//   PLC_TMO_VAC Instance <-> Device 1 (EtherCAT)/TMO_K4S2_DRL_02 (EK1100)/K4S2_02_E12 (EL2794)
//     PlcTask Outputs/GVL_Hutch_Pumps.PA1K4_IP1_PTM_01.q_RunDO <-> Channel 1/Output
//     PlcTask Outputs/GVL_Hutch_Pumps.PA1K4_IP1_PTM_02.q_RunDO <-> Channel 3/Output
//     PlcTask Outputs/GVL_Hutch_Pumps.PA1K4_IP1_PTM_01.q_xReset <-> Channel 2/Output
//     PlcTask Outputs/GVL_Hutch_Pumps.PA1K4_IP1_PTM_02.q_xReset <-> Channel 4/Output
//   PLC_TMO_VAC Instance <-> Device 1 (EtherCAT)/TMO_K4S2_DRL_02 (EK1100)/K4S2_02_E13 (EL1004)
//     PlcTask Inputs/GVL_Hutch_Pumps.PA1K4_IP1_PTM_03.i_xAtSpd <-> Channel 2/Input
//     PlcTask Inputs/GVL_Hutch_Pumps.PA1K4_IP1_PTM_03.i_xFaultNC <-> Channel 1/Input
//   PLC_TMO_VAC Instance <-> Device 1 (EtherCAT)/TMO_K4S2_DRL_02 (EK1100)/K4S2_02_E14 (EL2794)
//     PlcTask Outputs/GVL_Hutch_Pumps.PA1K4_IP1_PTM_03.q_RunDO <-> Channel 1/Output
//     PlcTask Outputs/GVL_Hutch_Pumps.PA1K4_IP1_PTM_03.q_xReset <-> Channel 2/Output
//   PLC_TMO_VAC Instance <-> Device 1 (EtherCAT)/TMO_K4S2_DRL_02 (EK1100)/K4S2_02_E15 (EL1004)
//     PlcTask Inputs/GVL_Hutch_Pumps.IM4K4_PPM_PTM_01.i_xAtSpd <-> Channel 2/Input
//     PlcTask Inputs/GVL_Hutch_Pumps.IM4K4_PPM_PTM_01.i_xFaultNC <-> Channel 1/Input
//     PlcTask Inputs/GVL_Hutch_Pumps.LI1K4_IP1_PTM_01.i_xAtSpd <-> Channel 4/Input
//     PlcTask Inputs/GVL_Hutch_Pumps.LI1K4_IP1_PTM_01.i_xFaultNC <-> Channel 3/Input
//   PLC_TMO_VAC Instance <-> Device 1 (EtherCAT)/TMO_K4S2_DRL_02 (EK1100)/K4S2_02_E16 (EL2794)
//     PlcTask Outputs/GVL_Hutch_Pumps.IM4K4_PPM_PTM_01.q_RunDO <-> Channel 1/Output
//     PlcTask Outputs/GVL_Hutch_Pumps.LI1K4_IP1_PTM_01.q_RunDO <-> Channel 2/Output
//   PLC_TMO_VAC Instance <-> Device 1 (EtherCAT)/TMO_K4S2_DRL_02 (EK1100)/K4S2_02_E17 (EL6001)
//     ComTask Inputs/GVL_COM.K4S2_02_E17_stComIn/D[0] <-> COM Inputs/Data In 0
//     ComTask Inputs/GVL_COM.K4S2_02_E17_stComIn/D[10] <-> COM Inputs/Data In 10
//     ComTask Inputs/GVL_COM.K4S2_02_E17_stComIn/D[11] <-> COM Inputs/Data In 11
//     ComTask Inputs/GVL_COM.K4S2_02_E17_stComIn/D[12] <-> COM Inputs/Data In 12
//     ComTask Inputs/GVL_COM.K4S2_02_E17_stComIn/D[13] <-> COM Inputs/Data In 13
//     ComTask Inputs/GVL_COM.K4S2_02_E17_stComIn/D[14] <-> COM Inputs/Data In 14
//     ComTask Inputs/GVL_COM.K4S2_02_E17_stComIn/D[15] <-> COM Inputs/Data In 15
//     ComTask Inputs/GVL_COM.K4S2_02_E17_stComIn/D[16] <-> COM Inputs/Data In 16
//     ComTask Inputs/GVL_COM.K4S2_02_E17_stComIn/D[17] <-> COM Inputs/Data In 17
//     ComTask Inputs/GVL_COM.K4S2_02_E17_stComIn/D[18] <-> COM Inputs/Data In 18
//     ComTask Inputs/GVL_COM.K4S2_02_E17_stComIn/D[19] <-> COM Inputs/Data In 19
//     ComTask Inputs/GVL_COM.K4S2_02_E17_stComIn/D[1] <-> COM Inputs/Data In 1
//     ComTask Inputs/GVL_COM.K4S2_02_E17_stComIn/D[20] <-> COM Inputs/Data In 20
//     ComTask Inputs/GVL_COM.K4S2_02_E17_stComIn/D[21] <-> COM Inputs/Data In 21
//     ComTask Inputs/GVL_COM.K4S2_02_E17_stComIn/D[2] <-> COM Inputs/Data In 2
//     ComTask Inputs/GVL_COM.K4S2_02_E17_stComIn/D[3] <-> COM Inputs/Data In 3
//     ComTask Inputs/GVL_COM.K4S2_02_E17_stComIn/D[4] <-> COM Inputs/Data In 4
//     ComTask Inputs/GVL_COM.K4S2_02_E17_stComIn/D[5] <-> COM Inputs/Data In 5
//     ComTask Inputs/GVL_COM.K4S2_02_E17_stComIn/D[6] <-> COM Inputs/Data In 6
//     ComTask Inputs/GVL_COM.K4S2_02_E17_stComIn/D[7] <-> COM Inputs/Data In 7
//     ComTask Inputs/GVL_COM.K4S2_02_E17_stComIn/D[8] <-> COM Inputs/Data In 8
//     ComTask Inputs/GVL_COM.K4S2_02_E17_stComIn/D[9] <-> COM Inputs/Data In 9
//     ComTask Inputs/GVL_COM.K4S2_02_E17_stComIn/Status <-> COM Inputs/Status
//     ComTask Outputs/GVL_COM.K4S2_02_E17_stComOut/Ctrl <-> COM Outputs/Ctrl
//     ComTask Outputs/GVL_COM.K4S2_02_E17_stComOut/D[0] <-> COM Outputs/Data Out 0
//     ComTask Outputs/GVL_COM.K4S2_02_E17_stComOut/D[10] <-> COM Outputs/Data Out 10
//     ComTask Outputs/GVL_COM.K4S2_02_E17_stComOut/D[11] <-> COM Outputs/Data Out 11
//     ComTask Outputs/GVL_COM.K4S2_02_E17_stComOut/D[12] <-> COM Outputs/Data Out 12
//     ComTask Outputs/GVL_COM.K4S2_02_E17_stComOut/D[13] <-> COM Outputs/Data Out 13
//     ComTask Outputs/GVL_COM.K4S2_02_E17_stComOut/D[14] <-> COM Outputs/Data Out 14
//     ComTask Outputs/GVL_COM.K4S2_02_E17_stComOut/D[15] <-> COM Outputs/Data Out 15
//     ComTask Outputs/GVL_COM.K4S2_02_E17_stComOut/D[16] <-> COM Outputs/Data Out 16
//     ComTask Outputs/GVL_COM.K4S2_02_E17_stComOut/D[17] <-> COM Outputs/Data Out 17
//     ComTask Outputs/GVL_COM.K4S2_02_E17_stComOut/D[18] <-> COM Outputs/Data Out 18
//     ComTask Outputs/GVL_COM.K4S2_02_E17_stComOut/D[19] <-> COM Outputs/Data Out 19
//     ComTask Outputs/GVL_COM.K4S2_02_E17_stComOut/D[1] <-> COM Outputs/Data Out 1
//     ComTask Outputs/GVL_COM.K4S2_02_E17_stComOut/D[20] <-> COM Outputs/Data Out 20
//     ComTask Outputs/GVL_COM.K4S2_02_E17_stComOut/D[21] <-> COM Outputs/Data Out 21
//     ComTask Outputs/GVL_COM.K4S2_02_E17_stComOut/D[2] <-> COM Outputs/Data Out 2
//     ComTask Outputs/GVL_COM.K4S2_02_E17_stComOut/D[3] <-> COM Outputs/Data Out 3
//     ComTask Outputs/GVL_COM.K4S2_02_E17_stComOut/D[4] <-> COM Outputs/Data Out 4
//     ComTask Outputs/GVL_COM.K4S2_02_E17_stComOut/D[5] <-> COM Outputs/Data Out 5
//     ComTask Outputs/GVL_COM.K4S2_02_E17_stComOut/D[6] <-> COM Outputs/Data Out 6
//     ComTask Outputs/GVL_COM.K4S2_02_E17_stComOut/D[7] <-> COM Outputs/Data Out 7
//     ComTask Outputs/GVL_COM.K4S2_02_E17_stComOut/D[8] <-> COM Outputs/Data Out 8
//     ComTask Outputs/GVL_COM.K4S2_02_E17_stComOut/D[9] <-> COM Outputs/Data Out 9
//   PLC_TMO_VAC Instance <-> Device 1 (EtherCAT)/TMO_K4S2_DRL_02 (EK1100)/K4S2_02_E18 (EL6001)
//     ComTask Inputs/GVL_COM.K4S2_02_E18_stComIn/D[0] <-> COM Inputs/Data In 0
//     ComTask Inputs/GVL_COM.K4S2_02_E18_stComIn/D[10] <-> COM Inputs/Data In 10
//     ComTask Inputs/GVL_COM.K4S2_02_E18_stComIn/D[11] <-> COM Inputs/Data In 11
//     ComTask Inputs/GVL_COM.K4S2_02_E18_stComIn/D[12] <-> COM Inputs/Data In 12
//     ComTask Inputs/GVL_COM.K4S2_02_E18_stComIn/D[13] <-> COM Inputs/Data In 13
//     ComTask Inputs/GVL_COM.K4S2_02_E18_stComIn/D[14] <-> COM Inputs/Data In 14
//     ComTask Inputs/GVL_COM.K4S2_02_E18_stComIn/D[15] <-> COM Inputs/Data In 15
//     ComTask Inputs/GVL_COM.K4S2_02_E18_stComIn/D[16] <-> COM Inputs/Data In 16
//     ComTask Inputs/GVL_COM.K4S2_02_E18_stComIn/D[17] <-> COM Inputs/Data In 17
//     ComTask Inputs/GVL_COM.K4S2_02_E18_stComIn/D[18] <-> COM Inputs/Data In 18
//     ComTask Inputs/GVL_COM.K4S2_02_E18_stComIn/D[19] <-> COM Inputs/Data In 19
//     ComTask Inputs/GVL_COM.K4S2_02_E18_stComIn/D[1] <-> COM Inputs/Data In 1
//     ComTask Inputs/GVL_COM.K4S2_02_E18_stComIn/D[20] <-> COM Inputs/Data In 20
//     ComTask Inputs/GVL_COM.K4S2_02_E18_stComIn/D[21] <-> COM Inputs/Data In 21
//     ComTask Inputs/GVL_COM.K4S2_02_E18_stComIn/D[2] <-> COM Inputs/Data In 2
//     ComTask Inputs/GVL_COM.K4S2_02_E18_stComIn/D[3] <-> COM Inputs/Data In 3
//     ComTask Inputs/GVL_COM.K4S2_02_E18_stComIn/D[4] <-> COM Inputs/Data In 4
//     ComTask Inputs/GVL_COM.K4S2_02_E18_stComIn/D[5] <-> COM Inputs/Data In 5
//     ComTask Inputs/GVL_COM.K4S2_02_E18_stComIn/D[6] <-> COM Inputs/Data In 6
//     ComTask Inputs/GVL_COM.K4S2_02_E18_stComIn/D[7] <-> COM Inputs/Data In 7
//     ComTask Inputs/GVL_COM.K4S2_02_E18_stComIn/D[8] <-> COM Inputs/Data In 8
//     ComTask Inputs/GVL_COM.K4S2_02_E18_stComIn/D[9] <-> COM Inputs/Data In 9
//     ComTask Inputs/GVL_COM.K4S2_02_E18_stComIn/Status <-> COM Inputs/Status
//     ComTask Outputs/GVL_COM.K4S2_02_E18_stComOut/Ctrl <-> COM Outputs/Ctrl
//     ComTask Outputs/GVL_COM.K4S2_02_E18_stComOut/D[0] <-> COM Outputs/Data Out 0
//     ComTask Outputs/GVL_COM.K4S2_02_E18_stComOut/D[10] <-> COM Outputs/Data Out 10
//     ComTask Outputs/GVL_COM.K4S2_02_E18_stComOut/D[11] <-> COM Outputs/Data Out 11
//     ComTask Outputs/GVL_COM.K4S2_02_E18_stComOut/D[12] <-> COM Outputs/Data Out 12
//     ComTask Outputs/GVL_COM.K4S2_02_E18_stComOut/D[13] <-> COM Outputs/Data Out 13
//     ComTask Outputs/GVL_COM.K4S2_02_E18_stComOut/D[14] <-> COM Outputs/Data Out 14
//     ComTask Outputs/GVL_COM.K4S2_02_E18_stComOut/D[15] <-> COM Outputs/Data Out 15
//     ComTask Outputs/GVL_COM.K4S2_02_E18_stComOut/D[16] <-> COM Outputs/Data Out 16
//     ComTask Outputs/GVL_COM.K4S2_02_E18_stComOut/D[17] <-> COM Outputs/Data Out 17
//     ComTask Outputs/GVL_COM.K4S2_02_E18_stComOut/D[18] <-> COM Outputs/Data Out 18
//     ComTask Outputs/GVL_COM.K4S2_02_E18_stComOut/D[19] <-> COM Outputs/Data Out 19
//     ComTask Outputs/GVL_COM.K4S2_02_E18_stComOut/D[1] <-> COM Outputs/Data Out 1
//     ComTask Outputs/GVL_COM.K4S2_02_E18_stComOut/D[20] <-> COM Outputs/Data Out 20
//     ComTask Outputs/GVL_COM.K4S2_02_E18_stComOut/D[21] <-> COM Outputs/Data Out 21
//     ComTask Outputs/GVL_COM.K4S2_02_E18_stComOut/D[2] <-> COM Outputs/Data Out 2
//     ComTask Outputs/GVL_COM.K4S2_02_E18_stComOut/D[3] <-> COM Outputs/Data Out 3
//     ComTask Outputs/GVL_COM.K4S2_02_E18_stComOut/D[4] <-> COM Outputs/Data Out 4
//     ComTask Outputs/GVL_COM.K4S2_02_E18_stComOut/D[5] <-> COM Outputs/Data Out 5
//     ComTask Outputs/GVL_COM.K4S2_02_E18_stComOut/D[6] <-> COM Outputs/Data Out 6
//     ComTask Outputs/GVL_COM.K4S2_02_E18_stComOut/D[7] <-> COM Outputs/Data Out 7
//     ComTask Outputs/GVL_COM.K4S2_02_E18_stComOut/D[8] <-> COM Outputs/Data Out 8
//     ComTask Outputs/GVL_COM.K4S2_02_E18_stComOut/D[9] <-> COM Outputs/Data Out 9
//   PLC_TMO_VAC Instance <-> Device 1 (EtherCAT)/TMO_K4S2_DRL_02 (EK1100)/K4S2_02_E19 (EL1004)
//     PlcTask Inputs/GVL_Hutch_Valves.TMO_ROUGH1_VRC_01.i_xClsLS <-> Channel 2/Input
//     PlcTask Inputs/GVL_Hutch_Valves.TMO_ROUGH2_VRC_01.i_xClsLS <-> Channel 4/Input
//     PlcTask Inputs/GVL_Hutch_Valves.TMO_ROUGH1_VRC_01.i_xOpnLS <-> Channel 1/Input
//     PlcTask Inputs/GVL_Hutch_Valves.TMO_ROUGH2_VRC_01.i_xOpnLS <-> Channel 3/Input
//   PLC_TMO_VAC Instance <-> Device 1 (EtherCAT)/TMO_K4S2_DRL_02 (EK1100)/K4S2_02_E2 (EL3174)
//     PlcTask Inputs/GVL_Hutch_Gauges.IM4K4_PPM_GCC_01.i_iPRESS_R <-> AI Standard Channel 2/Value
//     PlcTask Inputs/GVL_Hutch_Gauges.PA1K4_IP1_GPI_01.i_iPRESS_R <-> AI Standard Channel 1/Value
//   PLC_TMO_VAC Instance <-> Device 1 (EtherCAT)/TMO_K4S2_DRL_02 (EK1100)/K4S2_02_E20 (EL2004)
//     PlcTask Outputs/GVL_Hutch_Valves.TMO_ROUGH1_VRC_01.q_xOPN_DO <-> Channel 1/Output
//     PlcTask Outputs/GVL_Hutch_Valves.TMO_ROUGH2_VRC_01.q_xOPN_DO <-> Channel 2/Output
//     PlcTask Outputs/GVL_Variables.iHV_LOOP_FIM_ON <-> Channel 4/Output
//   PLC_TMO_VAC Instance <-> Device 1 (EtherCAT)/TMO_K4S2_DRL_02 (EK1100)/K4S2_02_E5 (EL2624)
//     PlcTask Outputs/GVL_Hutch_Gauges.IM4K4_PPM_GCC_01.q_xHV_DIS <-> Channel 4/Output
//     PlcTask Outputs/GVL_Hutch_Gauges.MR2K4_KBO_GCC_01.q_xHV_DIS <-> Channel 2/Output
//     PlcTask Outputs/GVL_Hutch_Gauges.PA1K4_IP1_GCC_01.q_xHV_DIS <-> Channel 3/Output
//   PLC_TMO_VAC Instance <-> Device 1 (EtherCAT)/TMO_K4S2_DRL_02 (EK1100)/K4S2_02_E7 (EL1124)
//     PlcTask Inputs/GVL_Hutch_Gauges.MR2K4_KBO_GCC_01.i_xDisc_Active <-> Channel 4/Input
//     PlcTask Inputs/GVL_Hutch_Gauges.MR2K4_KBO_GCC_01.i_xHV_ON <-> Channel 3/Input
//   PLC_TMO_VAC Instance <-> Device 1 (EtherCAT)/TMO_K4S6_ EP1 (EP4374-0002)
//     PlcTask Inputs/GVL_Hutch_Gauges.TMO_ROUGH1_GPI_03.i_iPRESS_R <-> AI Inputs Channel 1/Value
//     PlcTask Outputs/GVL_Hutch_Valves.TMO_ROUGH1_VFV_03.q_iRawPosition <-> AO Outputs Channel 3/Analog output
//   PLC_TMO_VAC Instance <-> Device 1 (EtherCAT)/TMO_K4S6_DRL_01 (EK1100)/K4S6_01_E1 (EL1004)
//     PlcTask Inputs/GVL_Hutch_Valves.TMO_ROUGH1_VRC_02.i_xClsLS <-> Channel 2/Input
//     PlcTask Inputs/GVL_Hutch_Valves.TMO_ROUGH1_VRC_02.i_xOpnLS <-> Channel 1/Input
//   PLC_TMO_VAC Instance <-> Device 1 (EtherCAT)/TMO_K4S6_DRL_01 (EK1100)/K4S6_01_E11 (EL1004)
//     PlcTask Inputs/GVL_Hutch_Pumps.IM5K4_PPM_PTM_01.i_xFaultNC <-> Channel 1/Input
//   PLC_TMO_VAC Instance <-> Device 1 (EtherCAT)/TMO_K4S6_DRL_01 (EK1100)/K4S6_01_E12 (EL2004)
//     PlcTask Outputs/GVL_Hutch_Pumps.IM5K4_PPM_PTM_01.q_PumpingStation <-> Channel 1/Output
//   PLC_TMO_VAC Instance <-> Device 1 (EtherCAT)/TMO_K4S6_DRL_01 (EK1100)/K4S6_01_E14 (EL2624)
//     PlcTask Outputs/GVL_Hutch_Gauges.IM5K4_PPM_GCC_01.q_xHV_DIS <-> Channel 2/Output
//     PlcTask Outputs/GVL_Hutch_Gauges.MR4K4_KBO_GCC_01.q_xHV_DIS <-> Channel 4/Output
//     PlcTask Outputs/GVL_Hutch_Gauges.PA2K4_IP1_GCC_01.q_xHV_DIS <-> Channel 3/Output
//     PlcTask Outputs/GVL_Hutch_Gauges.TM1K4_GCC_01.q_xHV_DIS <-> Channel 1/Output
//   PLC_TMO_VAC Instance <-> Device 1 (EtherCAT)/TMO_K4S6_DRL_01 (EK1100)/K4S6_01_E15 (EL3174)
//     PlcTask Inputs/GVL_Hutch_Gauges.IM5K4_PPM_GCC_01.i_iPRESS_R <-> AI Standard Channel 2/Value
//     PlcTask Inputs/GVL_Hutch_Gauges.PA2K4_IP1_GCC_01.i_iPRESS_R <-> AI Standard Channel 3/Value
//     PlcTask Inputs/GVL_Hutch_Gauges.PA2K4_IP1_GPI_01.i_iPRESS_R <-> AI Standard Channel 4/Value
//     PlcTask Inputs/GVL_Hutch_Gauges.TM1K4_GCC_01.i_iPRESS_R <-> AI Standard Channel 1/Value
//   PLC_TMO_VAC Instance <-> Device 1 (EtherCAT)/TMO_K4S6_DRL_01 (EK1100)/K4S6_01_E18 (EL3174)
//     PlcTask Inputs/GVL_Hutch_Gauges.IM5K4_PPM_GPI_01.i_iPRESS_R <-> AI Standard Channel 3/Value
//     PlcTask Inputs/GVL_Hutch_Gauges.MR4K4_KBO_GCC_01.i_iPRESS_R <-> AI Standard Channel 2/Value
//     PlcTask Inputs/GVL_Hutch_Gauges.MR4K4_KBO_GPI_01.i_iPRESS_R <-> AI Standard Channel 1/Value
//   PLC_TMO_VAC Instance <-> Device 1 (EtherCAT)/TMO_K4S6_DRL_01 (EK1100)/K4S6_01_E2 (EL2004)
//     PlcTask Outputs/GVL_Hutch_Valves.TMO_ROUGH1_VRC_02.q_xOPN_DO <-> Channel 1/Output
//   PLC_TMO_VAC Instance <-> Device 1 (EtherCAT)/TMO_K4S6_DRL_01 (EK1100)/K4S6_01_E20 (EL1124)
//     PlcTask Inputs/GVL_Hutch_Gauges.TM1K4_GCC_01.i_xDisc_Active <-> Channel 2/Input
//     PlcTask Inputs/GVL_Hutch_Gauges.TM1K4_GCC_01.i_xHV_ON <-> Channel 1/Input
//   PLC_TMO_VAC Instance <-> Device 1 (EtherCAT)/TMO_K4S6_DRL_01 (EK1100)/K4S6_01_E21 (EL1124)
//     PlcTask Inputs/GVL_Hutch_Gauges.MR4K4_KBO_GCC_01.i_xDisc_Active <-> Channel 4/Input
//     PlcTask Inputs/GVL_Hutch_Gauges.MR4K4_KBO_GCC_01.i_xHV_ON <-> Channel 3/Input
//     PlcTask Inputs/GVL_Hutch_Gauges.PA2K4_IP1_GCC_01.i_xDisc_Active <-> Channel 2/Input
//     PlcTask Inputs/GVL_Hutch_Gauges.PA2K4_IP1_GCC_01.i_xHV_ON <-> Channel 1/Input
//   PLC_TMO_VAC Instance <-> Device 1 (EtherCAT)/TMO_K4S6_DRL_01 (EK1100)/K4S6_01_E3 (EL1004)
//     PlcTask Inputs/GVL_Hutch_Valves.LI3K4_IP1_VWC_01.i_xClsLS <-> Channel 2/Input
//     PlcTask Inputs/GVL_Hutch_Valves.LI3K4_IP1_VWC_01.i_xOpnLS <-> Channel 1/Input
//     PlcTask Inputs/GVL_Hutch_Valves.PC5K4_VWC_01.i_xClsLS <-> Channel 4/Input
//     PlcTask Inputs/GVL_Hutch_Valves.PC5K4_VWC_01.i_xOpnLS <-> Channel 3/Input
//   PLC_TMO_VAC Instance <-> Device 1 (EtherCAT)/TMO_K4S6_DRL_01 (EK1100)/K4S6_01_E4 (EL2004)
//     PlcTask Outputs/GVL_Hutch_Valves.LI3K4_IP1_VWC_01.q_xOPN_DO <-> Channel 1/Output
//     PlcTask Outputs/GVL_Hutch_Valves.PC5K4_VWC_01.q_xOPN_DO <-> Channel 2/Output
//   PLC_TMO_VAC Instance <-> Device 1 (EtherCAT)/TMO_K4S6_DRL_01 (EK1100)/K4S6_01_E5 (EL6021)
//     ComTask Inputs/GVL_COM.K4S6_01_E5_stComIn/D[0] <-> COM TxPDO-Map Inputs/Data In 0
//     ComTask Inputs/GVL_COM.K4S6_01_E5_stComIn/D[10] <-> COM TxPDO-Map Inputs/Data In 10
//     ComTask Inputs/GVL_COM.K4S6_01_E5_stComIn/D[11] <-> COM TxPDO-Map Inputs/Data In 11
//     ComTask Inputs/GVL_COM.K4S6_01_E5_stComIn/D[12] <-> COM TxPDO-Map Inputs/Data In 12
//     ComTask Inputs/GVL_COM.K4S6_01_E5_stComIn/D[13] <-> COM TxPDO-Map Inputs/Data In 13
//     ComTask Inputs/GVL_COM.K4S6_01_E5_stComIn/D[14] <-> COM TxPDO-Map Inputs/Data In 14
//     ComTask Inputs/GVL_COM.K4S6_01_E5_stComIn/D[15] <-> COM TxPDO-Map Inputs/Data In 15
//     ComTask Inputs/GVL_COM.K4S6_01_E5_stComIn/D[16] <-> COM TxPDO-Map Inputs/Data In 16
//     ComTask Inputs/GVL_COM.K4S6_01_E5_stComIn/D[17] <-> COM TxPDO-Map Inputs/Data In 17
//     ComTask Inputs/GVL_COM.K4S6_01_E5_stComIn/D[18] <-> COM TxPDO-Map Inputs/Data In 18
//     ComTask Inputs/GVL_COM.K4S6_01_E5_stComIn/D[19] <-> COM TxPDO-Map Inputs/Data In 19
//     ComTask Inputs/GVL_COM.K4S6_01_E5_stComIn/D[1] <-> COM TxPDO-Map Inputs/Data In 1
//     ComTask Inputs/GVL_COM.K4S6_01_E5_stComIn/D[20] <-> COM TxPDO-Map Inputs/Data In 20
//     ComTask Inputs/GVL_COM.K4S6_01_E5_stComIn/D[21] <-> COM TxPDO-Map Inputs/Data In 21
//     ComTask Inputs/GVL_COM.K4S6_01_E5_stComIn/D[2] <-> COM TxPDO-Map Inputs/Data In 2
//     ComTask Inputs/GVL_COM.K4S6_01_E5_stComIn/D[3] <-> COM TxPDO-Map Inputs/Data In 3
//     ComTask Inputs/GVL_COM.K4S6_01_E5_stComIn/D[4] <-> COM TxPDO-Map Inputs/Data In 4
//     ComTask Inputs/GVL_COM.K4S6_01_E5_stComIn/D[5] <-> COM TxPDO-Map Inputs/Data In 5
//     ComTask Inputs/GVL_COM.K4S6_01_E5_stComIn/D[6] <-> COM TxPDO-Map Inputs/Data In 6
//     ComTask Inputs/GVL_COM.K4S6_01_E5_stComIn/D[7] <-> COM TxPDO-Map Inputs/Data In 7
//     ComTask Inputs/GVL_COM.K4S6_01_E5_stComIn/D[8] <-> COM TxPDO-Map Inputs/Data In 8
//     ComTask Inputs/GVL_COM.K4S6_01_E5_stComIn/D[9] <-> COM TxPDO-Map Inputs/Data In 9
//     ComTask Inputs/GVL_COM.K4S6_01_E5_stComIn/Status <-> COM TxPDO-Map Inputs/Status
//     ComTask Outputs/GVL_COM.K4S6_01_E5_stComOut/Ctrl <-> COM RxPDO-Map Outputs/Ctrl
//     ComTask Outputs/GVL_COM.K4S6_01_E5_stComOut/D[0] <-> COM RxPDO-Map Outputs/Data Out 0
//     ComTask Outputs/GVL_COM.K4S6_01_E5_stComOut/D[10] <-> COM RxPDO-Map Outputs/Data Out 10
//     ComTask Outputs/GVL_COM.K4S6_01_E5_stComOut/D[11] <-> COM RxPDO-Map Outputs/Data Out 11
//     ComTask Outputs/GVL_COM.K4S6_01_E5_stComOut/D[12] <-> COM RxPDO-Map Outputs/Data Out 12
//     ComTask Outputs/GVL_COM.K4S6_01_E5_stComOut/D[13] <-> COM RxPDO-Map Outputs/Data Out 13
//     ComTask Outputs/GVL_COM.K4S6_01_E5_stComOut/D[14] <-> COM RxPDO-Map Outputs/Data Out 14
//     ComTask Outputs/GVL_COM.K4S6_01_E5_stComOut/D[15] <-> COM RxPDO-Map Outputs/Data Out 15
//     ComTask Outputs/GVL_COM.K4S6_01_E5_stComOut/D[16] <-> COM RxPDO-Map Outputs/Data Out 16
//     ComTask Outputs/GVL_COM.K4S6_01_E5_stComOut/D[17] <-> COM RxPDO-Map Outputs/Data Out 17
//     ComTask Outputs/GVL_COM.K4S6_01_E5_stComOut/D[18] <-> COM RxPDO-Map Outputs/Data Out 18
//     ComTask Outputs/GVL_COM.K4S6_01_E5_stComOut/D[19] <-> COM RxPDO-Map Outputs/Data Out 19
//     ComTask Outputs/GVL_COM.K4S6_01_E5_stComOut/D[1] <-> COM RxPDO-Map Outputs/Data Out 1
//     ComTask Outputs/GVL_COM.K4S6_01_E5_stComOut/D[20] <-> COM RxPDO-Map Outputs/Data Out 20
//     ComTask Outputs/GVL_COM.K4S6_01_E5_stComOut/D[21] <-> COM RxPDO-Map Outputs/Data Out 21
//     ComTask Outputs/GVL_COM.K4S6_01_E5_stComOut/D[2] <-> COM RxPDO-Map Outputs/Data Out 2
//     ComTask Outputs/GVL_COM.K4S6_01_E5_stComOut/D[3] <-> COM RxPDO-Map Outputs/Data Out 3
//     ComTask Outputs/GVL_COM.K4S6_01_E5_stComOut/D[4] <-> COM RxPDO-Map Outputs/Data Out 4
//     ComTask Outputs/GVL_COM.K4S6_01_E5_stComOut/D[5] <-> COM RxPDO-Map Outputs/Data Out 5
//     ComTask Outputs/GVL_COM.K4S6_01_E5_stComOut/D[6] <-> COM RxPDO-Map Outputs/Data Out 6
//     ComTask Outputs/GVL_COM.K4S6_01_E5_stComOut/D[7] <-> COM RxPDO-Map Outputs/Data Out 7
//     ComTask Outputs/GVL_COM.K4S6_01_E5_stComOut/D[8] <-> COM RxPDO-Map Outputs/Data Out 8
//     ComTask Outputs/GVL_COM.K4S6_01_E5_stComOut/D[9] <-> COM RxPDO-Map Outputs/Data Out 9
//   PLC_TMO_VAC Instance <-> Device 1 (EtherCAT)/TMO_K4S6_DRL_01 (EK1100)/K4S6_01_E6 (EL1004)
//     PlcTask Inputs/GVL_Hutch_Pumps.LI3K4_IP1_OUT_PTM_01.i_xAtSpd <-> Channel 1/Input
//     PlcTask Inputs/GVL_Hutch_Pumps.LI3K4_IP1_OUT_PTM_01.i_xFaultNC <-> Channel 3/Input
//     PlcTask Inputs/GVL_Hutch_Pumps.LI3K4_IP1_OUT_PTM_01.i_xRemote <-> Channel 2/Input
//     PlcTask Inputs/GVL_Hutch_Pumps.TM1K4_PTM_01.i_xAtSpd <-> Channel 4/Input
//   PLC_TMO_VAC Instance <-> Device 1 (EtherCAT)/TMO_K4S6_DRL_01 (EK1100)/K4S6_01_E7 (EL2004)
//     PlcTask Outputs/GVL_Hutch_Pumps.LI3K4_IP1_OUT_PTM_01.q_PumpingStation <-> Channel 3/Output
//     PlcTask Outputs/GVL_Hutch_Pumps.LI3K4_IP1_OUT_PTM_01.q_RunDO <-> Channel 1/Output
//     PlcTask Outputs/GVL_Hutch_Pumps.LI3K4_IP1_OUT_PTM_01.q_xRemote <-> Channel 2/Output
//     PlcTask Outputs/GVL_Hutch_Pumps.TM1K4_PTM_01.q_RunDO <-> Channel 4/Output
//   PLC_TMO_VAC Instance <-> Device 1 (EtherCAT)/TMO_K4S6_DRL_01 (EK1100)/K4S6_01_E8 (EL1004)
//     PlcTask Inputs/GVL_Hutch_Pumps.IM5K4_PPM_PTM_01.i_xAtSpd <-> Channel 3/Input
//     PlcTask Inputs/GVL_Hutch_Pumps.IM5K4_PPM_PTM_01.i_xRemote <-> Channel 4/Input
//     PlcTask Inputs/GVL_Hutch_Pumps.TM1K4_PTM_01.i_xFaultNC <-> Channel 2/Input
//     PlcTask Inputs/GVL_Hutch_Pumps.TM1K4_PTM_01.i_xRemote <-> Channel 1/Input
//   PLC_TMO_VAC Instance <-> Device 1 (EtherCAT)/TMO_K4S6_DRL_01 (EK1100)/K4S6_01_E9 (EL2004)
//     PlcTask Outputs/GVL_Hutch_Pumps.IM5K4_PPM_PTM_01.q_RunDO <-> Channel 3/Output
//     PlcTask Outputs/GVL_Hutch_Pumps.IM5K4_PPM_PTM_01.q_xRemote <-> Channel 4/Output
//     PlcTask Outputs/GVL_Hutch_Pumps.TM1K4_PTM_01.q_PumpingStation <-> Channel 2/Output
//     PlcTask Outputs/GVL_Hutch_Pumps.TM1K4_PTM_01.q_xRemote <-> Channel 1/Output
//   PLC_TMO_VAC Instance <-> Device 1 (EtherCAT)/TMO_K4S8_DRL_01 (EK1100)/K4S8_01_E1 (EL1004)
//     FSVTask Inputs/GVL_FS_Devices.MR4K4_KBO_VFS_1.i_xClsLS <-> Channel 1/Input
//     FSVTask Inputs/GVL_FS_Devices.MR4K4_KBO_VFS_1.i_xOpnLS <-> Channel 2/Input
//   PLC_TMO_VAC Instance <-> Device 1 (EtherCAT)/TMO_K4S8_DRL_01 (EK1100)/K4S8_01_E3 (EL2202)
//     FSVTask Outputs/GVL_FS_Devices.MR4K4_KBO_VFS_1.q_xClose_A <-> Channel 1/Output
//     FSVTask Outputs/GVL_FS_Devices.MR4K4_KBO_VFS_1.q_xClose_B <-> Channel 2/Output
//   PLC_TMO_VAC Instance <-> Device 1 (EtherCAT)/TMO_K4S8_DRL_01 (EK1100)/K4S8_01_E4 (EL2202)
//     FSVTask Outputs/GVL_FS_Devices.MR4K4_KBO_VFS_1.q_xClose_C <-> Channel 1/Output
//     FSVTask Outputs/GVL_FS_Devices.MR4K4_KBO_VFS_1.q_xOPN_DO <-> Channel 2/Output
//   PLC_TMO_VAC Instance <-> Device 1 (EtherCAT)/TMO_K4S8_DRL_01 (EK1100)/K4S8_01_E5 (EL1004)
//     PlcTask Inputs/GVL_Hutch_Valves.MR4K4_KBO_VWC_01.i_xClsLS <-> Channel 2/Input
//     PlcTask Inputs/GVL_Hutch_Valves.MR5K4_KBO_VWC_01.i_xClsLS <-> Channel 4/Input
//     PlcTask Inputs/GVL_Hutch_Valves.MR4K4_KBO_VWC_01.i_xOpnLS <-> Channel 1/Input
//     PlcTask Inputs/GVL_Hutch_Valves.MR5K4_KBO_VWC_01.i_xOpnLS <-> Channel 3/Input
//   PLC_TMO_VAC Instance <-> Device 1 (EtherCAT)/TMO_K4S8_DRL_01 (EK1100)/K4S8_01_E6 (EL2004)
//     PlcTask Outputs/GVL_Hutch_Valves.MR4K4_KBO_VWC_01.q_xOPN_DO <-> Channel 1/Output
//     PlcTask Outputs/GVL_Hutch_Valves.MR5K4_KBO_VWC_01.q_xOPN_DO <-> Channel 2/Output
//   PLC_TMO_VAC Instance <-> Device 1 (EtherCAT)/TMO_K4S8_DRL_02 (EK1100)/K4S8_02_E1 (EL1004)
//     PlcTask Inputs/GVL_Hutch_Valves.TM2K4_KBO_VWC_01.i_xClsLS <-> Channel 2/Input
//     PlcTask Inputs/GVL_Hutch_Valves.TM2K4_KBO_VWC_01.i_xOpnLS <-> Channel 1/Input
//   PLC_TMO_VAC Instance <-> Device 1 (EtherCAT)/TMO_K4S8_DRL_02 (EK1100)/K4S8_02_E2 (EL2004)
//     PlcTask Outputs/GVL_Hutch_Valves.TM2K4_KBO_VWC_01.q_xOPN_DO <-> Channel 1/Output
//   PLC_TMO_VAC Instance <-> Device 1 (EtherCAT)/TMO_K4S8_DRL_02 (EK1100)/K4S8_02_E3 (EL2624)
//     PlcTask Outputs/GVL_Hutch_Gauges.PF2K4_WFS_GCC_01.q_xHV_DIS <-> Channel 2/Output
//     PlcTask Outputs/GVL_Hutch_Gauges.TM2K4_KBO_GCC_01.q_xHV_DIS <-> Channel 1/Output
//   PLC_TMO_VAC Instance <-> Device 1 (EtherCAT)/TMO_K4S8_DRL_02 (EK1100)/K4S8_02_E4 (EL3174)
//     PlcTask Inputs/GVL_Hutch_Gauges.PF2K4_WFS_GCC_01.i_iPRESS_R <-> AI Standard Channel 2/Value
//     PlcTask Inputs/GVL_Hutch_Gauges.TM2K4_KBO_GCC_01.i_iPRESS_R <-> AI Standard Channel 1/Value
//     PlcTask Inputs/GVL_Hutch_Gauges.TM2K4_KBO_GPI_01.i_iPRESS_R <-> AI Standard Channel 3/Value
//   PLC_TMO_VAC Instance <-> Device 1 (EtherCAT)/TMO_K4S8_DRL_02 (EK1100)/K4S8_02_E8 (EL1124)
//     PlcTask Inputs/GVL_Hutch_Gauges.TM2K4_KBO_GCC_01.i_xDisc_Active <-> Channel 2/Input
//     PlcTask Inputs/GVL_Hutch_Gauges.TM2K4_KBO_GCC_01.i_xHV_ON <-> Channel 1/Input
//   PLC_TMO_VAC Instance <-> Device 1 (EtherCAT)/TMO_WALL_WEST_EP01 (EP4374-0002)
//     PlcTask Inputs/GVL_Hutch_Gauges.TMO_ROUGH1_GPI_01.i_iPRESS_R <-> AI Inputs Channel 1/Value
//     PlcTask Inputs/GVL_Hutch_Gauges.TMO_ROUGH2_GPI_01.i_iPRESS_R <-> AI Inputs Channel 2/Value
//     PlcTask Outputs/GVL_Hutch_Valves.TMO_ROUGH1_VFV_01.q_iRawPosition <-> AO Outputs Channel 3/Analog output
//   PLC_TMO_VAC Instance <-> PLC_TMO_VAC/PLC_TMO_VAC Instance
//     FSVTask Inputs/GVL_FS_Devices.MR3K4_KBO_VFS_1.i_ResetFaultCounter <-> PlcTask Outputs/GVL_FS_Devices.MR3K4_KBO_VFS_Interface.q_ResetFaultCounter
//     FSVTask Inputs/GVL_FS_Devices.MR4K4_KBO_VFS_1.i_ResetFaultCounter <-> PlcTask Outputs/GVL_FS_Devices.MR4K4_KBO_VFS_Interface.q_ResetFaultCounter
//     FSVTask Inputs/GVL_FS_Devices.MR3K4_KBO_VFS_1.i_e2OO3_MODE <-> PlcTask Outputs/GVL_FS_Devices.MR3K4_KBO_VFS_Interface.q_e2OO3_MODE
//     FSVTask Inputs/GVL_FS_Devices.MR4K4_KBO_VFS_1.i_e2OO3_MODE <-> PlcTask Outputs/GVL_FS_Devices.MR4K4_KBO_VFS_Interface.q_e2OO3_MODE
//     FSVTask Inputs/GVL_FS_Devices.MR3K4_KBO_VFS_1.i_xCLS_SW <-> PlcTask Outputs/GVL_FS_Devices.MR3K4_KBO_VFS_Interface.q_xCLS_SW
//     FSVTask Inputs/GVL_FS_Devices.MR4K4_KBO_VFS_1.i_xCLS_SW <-> PlcTask Outputs/GVL_FS_Devices.MR4K4_KBO_VFS_Interface.q_xCLS_SW
//     FSVTask Inputs/GVL_FS_Devices.MR3K4_KBO_VFS_1.i_xOPN_SW <-> PlcTask Outputs/GVL_FS_Devices.MR3K4_KBO_VFS_Interface.q_xOPN_SW
//     FSVTask Inputs/GVL_FS_Devices.MR4K4_KBO_VFS_1.i_xOPN_SW <-> PlcTask Outputs/GVL_FS_Devices.MR4K4_KBO_VFS_Interface.q_xOPN_SW
//     FSVTask Inputs/GVL_FS_Devices.MR3K4_KBO_VFS_1.i_xOverrideMode <-> PlcTask Outputs/GVL_FS_Devices.MR3K4_KBO_VFS_Interface.q_xOverrideMode
//     FSVTask Inputs/GVL_FS_Devices.MR4K4_KBO_VFS_1.i_xOverrideMode <-> PlcTask Outputs/GVL_FS_Devices.MR4K4_KBO_VFS_Interface.q_xOverrideMode
//     FSVTask Inputs/GVL_FS_Devices.MR3K4_KBO_VFS_1.i_xOverrideOpen <-> PlcTask Outputs/GVL_FS_Devices.MR3K4_KBO_VFS_Interface.q_xOverrideOpen
//     FSVTask Inputs/GVL_FS_Devices.MR4K4_KBO_VFS_1.i_xOverrideOpen <-> PlcTask Outputs/GVL_FS_Devices.MR4K4_KBO_VFS_Interface.q_xOverrideOpen
//     FSVTask Inputs/GVL_FS_Devices.MR3K4_KBO_VFS_1.i_xPress_OK_IG1 <-> PlcTask Outputs/GVL_FS_Devices.MR3K4_KBO_VFS_Interface.q_xPRESS_OK_IG1
//     FSVTask Inputs/GVL_FS_Devices.MR3K4_KBO_VFS_1.i_xPress_OK_IG2 <-> PlcTask Outputs/GVL_FS_Devices.MR3K4_KBO_VFS_Interface.q_xPRESS_OK_IG2
//     FSVTask Inputs/GVL_FS_Devices.MR3K4_KBO_VFS_1.i_xPress_OK_IG3 <-> PlcTask Outputs/GVL_FS_Devices.MR3K4_KBO_VFS_Interface.q_xPRESS_OK_IG3
//     FSVTask Inputs/GVL_FS_Devices.MR4K4_KBO_VFS_1.i_xPress_OK_IG1 <-> PlcTask Outputs/GVL_FS_Devices.MR4K4_KBO_VFS_Interface.q_xPRESS_OK_IG1
//     FSVTask Inputs/GVL_FS_Devices.MR4K4_KBO_VFS_1.i_xPress_OK_IG2 <-> PlcTask Outputs/GVL_FS_Devices.MR4K4_KBO_VFS_Interface.q_xPRESS_OK_IG2
//     FSVTask Inputs/GVL_FS_Devices.MR4K4_KBO_VFS_1.i_xPress_OK_IG3 <-> PlcTask Outputs/GVL_FS_Devices.MR4K4_KBO_VFS_Interface.q_xPRESS_OK_IG3
//     FSVTask Inputs/GVL_FS_Devices.MR3K4_KBO_VFS_1.i_xVAC_FAULT_Reset <-> PlcTask Outputs/GVL_FS_Devices.MR3K4_KBO_VFS_Interface.q_xVAC_FAULT_Reset
//     FSVTask Inputs/GVL_FS_Devices.MR4K4_KBO_VFS_1.i_xVAC_FAULT_Reset <-> PlcTask Outputs/GVL_FS_Devices.MR4K4_KBO_VFS_Interface.q_xVAC_FAULT_Reset
//     FSVTask Inputs/GVL_FS_Devices.MR3K4_KBO_VFS_1.i_xVetoValveClosed <-> PlcTask Outputs/GVL_FS_Devices.MR3K4_KBO_VFS_Interface.q_xVetoValveClosed
//     FSVTask Inputs/GVL_FS_Devices.MR4K4_KBO_VFS_1.i_xVetoValveClosed <-> PlcTask Outputs/GVL_FS_Devices.MR4K4_KBO_VFS_Interface.q_xVetoValveClosed
//     FSVTask Inputs/GVL_FS_Devices.MR3K4_KBO_VFS_1.i_xVetoValveOpenDO <-> PlcTask Outputs/GVL_FS_Devices.MR3K4_KBO_VFS_Interface.q_xVetoValveOpenDO
//     FSVTask Inputs/GVL_FS_Devices.MR4K4_KBO_VFS_1.i_xVetoValveOpenDO <-> PlcTask Outputs/GVL_FS_Devices.MR4K4_KBO_VFS_Interface.q_xVetoValveOpenDO
//     FSVTask Inputs/GVL_FS_Devices.TV1K4_VFS_1.i_ResetFaultCounter <-> PlcTask Outputs/GVL_FS_Devices.TV1K4_VFS_Interface.q_ResetFaultCounter
//     FSVTask Inputs/GVL_FS_Devices.TV1K4_VFS_1.i_e2OO3_MODE <-> PlcTask Outputs/GVL_FS_Devices.TV1K4_VFS_Interface.q_e2OO3_MODE
//     FSVTask Inputs/GVL_FS_Devices.TV1K4_VFS_1.i_xCLS_SW <-> PlcTask Outputs/GVL_FS_Devices.TV1K4_VFS_Interface.q_xCLS_SW
//     FSVTask Inputs/GVL_FS_Devices.TV1K4_VFS_1.i_xOPN_SW <-> PlcTask Outputs/GVL_FS_Devices.TV1K4_VFS_Interface.q_xOPN_SW
//     FSVTask Inputs/GVL_FS_Devices.TV1K4_VFS_1.i_xOverrideMode <-> PlcTask Outputs/GVL_FS_Devices.TV1K4_VFS_Interface.q_xOverrideMode
//     FSVTask Inputs/GVL_FS_Devices.TV1K4_VFS_1.i_xOverrideOpen <-> PlcTask Outputs/GVL_FS_Devices.TV1K4_VFS_Interface.q_xOverrideOpen
//     FSVTask Inputs/GVL_FS_Devices.TV1K4_VFS_1.i_xPress_OK_IG1 <-> PlcTask Outputs/GVL_FS_Devices.TV1K4_VFS_Interface.q_xPRESS_OK_IG1
//     FSVTask Inputs/GVL_FS_Devices.TV1K4_VFS_1.i_xPress_OK_IG2 <-> PlcTask Outputs/GVL_FS_Devices.TV1K4_VFS_Interface.q_xPRESS_OK_IG2
//     FSVTask Inputs/GVL_FS_Devices.TV1K4_VFS_1.i_xPress_OK_IG3 <-> PlcTask Outputs/GVL_FS_Devices.TV1K4_VFS_Interface.q_xPRESS_OK_IG3
//     FSVTask Inputs/GVL_FS_Devices.TV1K4_VFS_1.i_xVAC_FAULT_Reset <-> PlcTask Outputs/GVL_FS_Devices.TV1K4_VFS_Interface.q_xVAC_FAULT_Reset
//     FSVTask Inputs/GVL_FS_Devices.TV1K4_VFS_1.i_xVetoValveClosed <-> PlcTask Outputs/GVL_FS_Devices.TV1K4_VFS_Interface.q_xVetoValveClosed
//     FSVTask Inputs/GVL_FS_Devices.TV1K4_VFS_1.i_xVetoValveOpenDO <-> PlcTask Outputs/GVL_FS_Devices.TV1K4_VFS_Interface.q_xVetoValveOpenDO
//     FSVTask Outputs/GVL_FS_Devices.MR3K4_KBO_VFS_1.q_eVFS_State <-> PlcTask Inputs/GVL_FS_Devices.MR3K4_KBO_VFS_Interface.i_eVFS_State
//     FSVTask Outputs/GVL_FS_Devices.MR4K4_KBO_VFS_1.q_eVFS_State <-> PlcTask Inputs/GVL_FS_Devices.MR4K4_KBO_VFS_Interface.i_eVFS_State
//     FSVTask Outputs/GVL_FS_Devices.MR3K4_KBO_VFS_1.q_nFltCount_IG1 <-> PlcTask Inputs/GVL_FS_Devices.MR3K4_KBO_VFS_Interface.i_nFltCount_IG1
//     FSVTask Outputs/GVL_FS_Devices.MR3K4_KBO_VFS_1.q_nFltCount_IG2 <-> PlcTask Inputs/GVL_FS_Devices.MR3K4_KBO_VFS_Interface.i_nFltCount_IG2
//     FSVTask Outputs/GVL_FS_Devices.MR3K4_KBO_VFS_1.q_nFltCount_IG3 <-> PlcTask Inputs/GVL_FS_Devices.MR3K4_KBO_VFS_Interface.i_nFltCount_IG3
//     FSVTask Outputs/GVL_FS_Devices.MR4K4_KBO_VFS_1.q_nFltCount_IG1 <-> PlcTask Inputs/GVL_FS_Devices.MR4K4_KBO_VFS_Interface.i_nFltCount_IG1
//     FSVTask Outputs/GVL_FS_Devices.MR4K4_KBO_VFS_1.q_nFltCount_IG2 <-> PlcTask Inputs/GVL_FS_Devices.MR4K4_KBO_VFS_Interface.i_nFltCount_IG2
//     FSVTask Outputs/GVL_FS_Devices.MR4K4_KBO_VFS_1.q_nFltCount_IG3 <-> PlcTask Inputs/GVL_FS_Devices.MR4K4_KBO_VFS_Interface.i_nFltCount_IG3
//     FSVTask Outputs/GVL_FS_Devices.MR3K4_KBO_VFS_1.q_xMPS_OK <-> PlcTask Inputs/GVL_FS_Devices.MR3K4_KBO_VFS_Interface.i_xMPS_OK
//     FSVTask Outputs/GVL_FS_Devices.MR4K4_KBO_VFS_1.q_xMPS_OK <-> PlcTask Inputs/GVL_FS_Devices.MR4K4_KBO_VFS_Interface.i_xMPS_OK
//     FSVTask Outputs/GVL_FS_Devices.MR3K4_KBO_VFS_1.q_xTrigger <-> PlcTask Inputs/GVL_FS_Devices.MR3K4_KBO_VFS_Interface.i_xTrigger
//     FSVTask Outputs/GVL_FS_Devices.MR4K4_KBO_VFS_1.q_xTrigger <-> PlcTask Inputs/GVL_FS_Devices.MR4K4_KBO_VFS_Interface.i_xTrigger
//     FSVTask Outputs/GVL_FS_Devices.MR3K4_KBO_VFS_1.q_xVAC_FAULT_OK <-> PlcTask Inputs/GVL_FS_Devices.MR3K4_KBO_VFS_Interface.i_xVAC_FAULT_OK
//     FSVTask Outputs/GVL_FS_Devices.MR4K4_KBO_VFS_1.q_xVAC_FAULT_OK <-> PlcTask Inputs/GVL_FS_Devices.MR4K4_KBO_VFS_Interface.i_xVAC_FAULT_OK
//     FSVTask Outputs/GVL_FS_Devices.MR3K4_KBO_VFS_1.q_xVFS_Closed <-> PlcTask Inputs/GVL_FS_Devices.MR3K4_KBO_VFS_Interface.i_xVFS_Closed
//     FSVTask Outputs/GVL_FS_Devices.MR4K4_KBO_VFS_1.q_xVFS_Closed <-> PlcTask Inputs/GVL_FS_Devices.MR4K4_KBO_VFS_Interface.i_xVFS_Closed
//     FSVTask Outputs/GVL_FS_Devices.MR3K4_KBO_VFS_1.q_xVFS_Open <-> PlcTask Inputs/GVL_FS_Devices.MR3K4_KBO_VFS_Interface.i_xVFS_Open
//     FSVTask Outputs/GVL_FS_Devices.MR4K4_KBO_VFS_1.q_xVFS_Open <-> PlcTask Inputs/GVL_FS_Devices.MR4K4_KBO_VFS_Interface.i_xVFS_Open
//     FSVTask Outputs/GVL_FS_Devices.TV1K4_VFS_1.q_eVFS_State <-> PlcTask Inputs/GVL_FS_Devices.TV1K4_VFS_Interface.i_eVFS_State
//     FSVTask Outputs/GVL_FS_Devices.TV1K4_VFS_1.q_nFltCount_IG1 <-> PlcTask Inputs/GVL_FS_Devices.TV1K4_VFS_Interface.i_nFltCount_IG1
//     FSVTask Outputs/GVL_FS_Devices.TV1K4_VFS_1.q_nFltCount_IG2 <-> PlcTask Inputs/GVL_FS_Devices.TV1K4_VFS_Interface.i_nFltCount_IG2
//     FSVTask Outputs/GVL_FS_Devices.TV1K4_VFS_1.q_nFltCount_IG3 <-> PlcTask Inputs/GVL_FS_Devices.TV1K4_VFS_Interface.i_nFltCount_IG3
//     FSVTask Outputs/GVL_FS_Devices.TV1K4_VFS_1.q_xMPS_OK <-> PlcTask Inputs/GVL_FS_Devices.TV1K4_VFS_Interface.i_xMPS_OK
//     FSVTask Outputs/GVL_FS_Devices.TV1K4_VFS_1.q_xTrigger <-> PlcTask Inputs/GVL_FS_Devices.TV1K4_VFS_Interface.i_xTrigger
//     FSVTask Outputs/GVL_FS_Devices.TV1K4_VFS_1.q_xVAC_FAULT_OK <-> PlcTask Inputs/GVL_FS_Devices.TV1K4_VFS_Interface.i_xVAC_FAULT_OK
//     FSVTask Outputs/GVL_FS_Devices.TV1K4_VFS_1.q_xVFS_Closed <-> PlcTask Inputs/GVL_FS_Devices.TV1K4_VFS_Interface.i_xVFS_Closed
//     FSVTask Outputs/GVL_FS_Devices.TV1K4_VFS_1.q_xVFS_Open <-> PlcTask Inputs/GVL_FS_Devices.TV1K4_VFS_Interface.i_xVFS_Open
//     PlcTask Inputs/GVL_FS_Devices.MR3K4_KBO_VFS_Interface.i_eVFS_State <-> FSVTask Outputs/GVL_FS_Devices.MR3K4_KBO_VFS_1.q_eVFS_State
//     PlcTask Inputs/GVL_FS_Devices.MR4K4_KBO_VFS_Interface.i_eVFS_State <-> FSVTask Outputs/GVL_FS_Devices.MR4K4_KBO_VFS_1.q_eVFS_State
//     PlcTask Inputs/GVL_FS_Devices.MR3K4_KBO_VFS_Interface.i_nFltCount_IG1 <-> FSVTask Outputs/GVL_FS_Devices.MR3K4_KBO_VFS_1.q_nFltCount_IG1
//     PlcTask Inputs/GVL_FS_Devices.MR3K4_KBO_VFS_Interface.i_nFltCount_IG2 <-> FSVTask Outputs/GVL_FS_Devices.MR3K4_KBO_VFS_1.q_nFltCount_IG2
//     PlcTask Inputs/GVL_FS_Devices.MR3K4_KBO_VFS_Interface.i_nFltCount_IG3 <-> FSVTask Outputs/GVL_FS_Devices.MR3K4_KBO_VFS_1.q_nFltCount_IG3
//     PlcTask Inputs/GVL_FS_Devices.MR4K4_KBO_VFS_Interface.i_nFltCount_IG1 <-> FSVTask Outputs/GVL_FS_Devices.MR4K4_KBO_VFS_1.q_nFltCount_IG1
//     PlcTask Inputs/GVL_FS_Devices.MR4K4_KBO_VFS_Interface.i_nFltCount_IG2 <-> FSVTask Outputs/GVL_FS_Devices.MR4K4_KBO_VFS_1.q_nFltCount_IG2
//     PlcTask Inputs/GVL_FS_Devices.MR4K4_KBO_VFS_Interface.i_nFltCount_IG3 <-> FSVTask Outputs/GVL_FS_Devices.MR4K4_KBO_VFS_1.q_nFltCount_IG3
//     PlcTask Inputs/GVL_FS_Devices.MR3K4_KBO_VFS_Interface.i_xMPS_OK <-> FSVTask Outputs/GVL_FS_Devices.MR3K4_KBO_VFS_1.q_xMPS_OK
//     PlcTask Inputs/GVL_FS_Devices.MR4K4_KBO_VFS_Interface.i_xMPS_OK <-> FSVTask Outputs/GVL_FS_Devices.MR4K4_KBO_VFS_1.q_xMPS_OK
//     PlcTask Inputs/GVL_FS_Devices.MR3K4_KBO_VFS_Interface.i_xTrigger <-> FSVTask Outputs/GVL_FS_Devices.MR3K4_KBO_VFS_1.q_xTrigger
//     PlcTask Inputs/GVL_FS_Devices.MR4K4_KBO_VFS_Interface.i_xTrigger <-> FSVTask Outputs/GVL_FS_Devices.MR4K4_KBO_VFS_1.q_xTrigger
//     PlcTask Inputs/GVL_FS_Devices.MR3K4_KBO_VFS_Interface.i_xVAC_FAULT_OK <-> FSVTask Outputs/GVL_FS_Devices.MR3K4_KBO_VFS_1.q_xVAC_FAULT_OK
//     PlcTask Inputs/GVL_FS_Devices.MR4K4_KBO_VFS_Interface.i_xVAC_FAULT_OK <-> FSVTask Outputs/GVL_FS_Devices.MR4K4_KBO_VFS_1.q_xVAC_FAULT_OK
//     PlcTask Inputs/GVL_FS_Devices.MR3K4_KBO_VFS_Interface.i_xVFS_Closed <-> FSVTask Outputs/GVL_FS_Devices.MR3K4_KBO_VFS_1.q_xVFS_Closed
//     PlcTask Inputs/GVL_FS_Devices.MR4K4_KBO_VFS_Interface.i_xVFS_Closed <-> FSVTask Outputs/GVL_FS_Devices.MR4K4_KBO_VFS_1.q_xVFS_Closed
//     PlcTask Inputs/GVL_FS_Devices.MR3K4_KBO_VFS_Interface.i_xVFS_Open <-> FSVTask Outputs/GVL_FS_Devices.MR3K4_KBO_VFS_1.q_xVFS_Open
//     PlcTask Inputs/GVL_FS_Devices.MR4K4_KBO_VFS_Interface.i_xVFS_Open <-> FSVTask Outputs/GVL_FS_Devices.MR4K4_KBO_VFS_1.q_xVFS_Open
//     PlcTask Inputs/GVL_FS_Devices.TV1K4_VFS_Interface.i_eVFS_State <-> FSVTask Outputs/GVL_FS_Devices.TV1K4_VFS_1.q_eVFS_State
//     PlcTask Inputs/GVL_FS_Devices.TV1K4_VFS_Interface.i_nFltCount_IG1 <-> FSVTask Outputs/GVL_FS_Devices.TV1K4_VFS_1.q_nFltCount_IG1
//     PlcTask Inputs/GVL_FS_Devices.TV1K4_VFS_Interface.i_nFltCount_IG2 <-> FSVTask Outputs/GVL_FS_Devices.TV1K4_VFS_1.q_nFltCount_IG2
//     PlcTask Inputs/GVL_FS_Devices.TV1K4_VFS_Interface.i_nFltCount_IG3 <-> FSVTask Outputs/GVL_FS_Devices.TV1K4_VFS_1.q_nFltCount_IG3
//     PlcTask Inputs/GVL_FS_Devices.TV1K4_VFS_Interface.i_xMPS_OK <-> FSVTask Outputs/GVL_FS_Devices.TV1K4_VFS_1.q_xMPS_OK
//     PlcTask Inputs/GVL_FS_Devices.TV1K4_VFS_Interface.i_xTrigger <-> FSVTask Outputs/GVL_FS_Devices.TV1K4_VFS_1.q_xTrigger
//     PlcTask Inputs/GVL_FS_Devices.TV1K4_VFS_Interface.i_xVAC_FAULT_OK <-> FSVTask Outputs/GVL_FS_Devices.TV1K4_VFS_1.q_xVAC_FAULT_OK
//     PlcTask Inputs/GVL_FS_Devices.TV1K4_VFS_Interface.i_xVFS_Closed <-> FSVTask Outputs/GVL_FS_Devices.TV1K4_VFS_1.q_xVFS_Closed
//     PlcTask Inputs/GVL_FS_Devices.TV1K4_VFS_Interface.i_xVFS_Open <-> FSVTask Outputs/GVL_FS_Devices.TV1K4_VFS_1.q_xVFS_Open
//     PlcTask Outputs/GVL_FS_Devices.MR3K4_KBO_VFS_Interface.q_ResetFaultCounter <-> FSVTask Inputs/GVL_FS_Devices.MR3K4_KBO_VFS_1.i_ResetFaultCounter
//     PlcTask Outputs/GVL_FS_Devices.MR4K4_KBO_VFS_Interface.q_ResetFaultCounter <-> FSVTask Inputs/GVL_FS_Devices.MR4K4_KBO_VFS_1.i_ResetFaultCounter
//     PlcTask Outputs/GVL_FS_Devices.MR3K4_KBO_VFS_Interface.q_e2OO3_MODE <-> FSVTask Inputs/GVL_FS_Devices.MR3K4_KBO_VFS_1.i_e2OO3_MODE
//     PlcTask Outputs/GVL_FS_Devices.MR4K4_KBO_VFS_Interface.q_e2OO3_MODE <-> FSVTask Inputs/GVL_FS_Devices.MR4K4_KBO_VFS_1.i_e2OO3_MODE
//     PlcTask Outputs/GVL_FS_Devices.MR3K4_KBO_VFS_Interface.q_xCLS_SW <-> FSVTask Inputs/GVL_FS_Devices.MR3K4_KBO_VFS_1.i_xCLS_SW
//     PlcTask Outputs/GVL_FS_Devices.MR4K4_KBO_VFS_Interface.q_xCLS_SW <-> FSVTask Inputs/GVL_FS_Devices.MR4K4_KBO_VFS_1.i_xCLS_SW
//     PlcTask Outputs/GVL_FS_Devices.MR3K4_KBO_VFS_Interface.q_xOPN_SW <-> FSVTask Inputs/GVL_FS_Devices.MR3K4_KBO_VFS_1.i_xOPN_SW
//     PlcTask Outputs/GVL_FS_Devices.MR4K4_KBO_VFS_Interface.q_xOPN_SW <-> FSVTask Inputs/GVL_FS_Devices.MR4K4_KBO_VFS_1.i_xOPN_SW
//     PlcTask Outputs/GVL_FS_Devices.MR3K4_KBO_VFS_Interface.q_xOverrideMode <-> FSVTask Inputs/GVL_FS_Devices.MR3K4_KBO_VFS_1.i_xOverrideMode
//     PlcTask Outputs/GVL_FS_Devices.MR4K4_KBO_VFS_Interface.q_xOverrideMode <-> FSVTask Inputs/GVL_FS_Devices.MR4K4_KBO_VFS_1.i_xOverrideMode
//     PlcTask Outputs/GVL_FS_Devices.MR3K4_KBO_VFS_Interface.q_xOverrideOpen <-> FSVTask Inputs/GVL_FS_Devices.MR3K4_KBO_VFS_1.i_xOverrideOpen
//     PlcTask Outputs/GVL_FS_Devices.MR4K4_KBO_VFS_Interface.q_xOverrideOpen <-> FSVTask Inputs/GVL_FS_Devices.MR4K4_KBO_VFS_1.i_xOverrideOpen
//     PlcTask Outputs/GVL_FS_Devices.MR3K4_KBO_VFS_Interface.q_xPRESS_OK_IG1 <-> FSVTask Inputs/GVL_FS_Devices.MR3K4_KBO_VFS_1.i_xPress_OK_IG1
//     PlcTask Outputs/GVL_FS_Devices.MR3K4_KBO_VFS_Interface.q_xPRESS_OK_IG2 <-> FSVTask Inputs/GVL_FS_Devices.MR3K4_KBO_VFS_1.i_xPress_OK_IG2
//     PlcTask Outputs/GVL_FS_Devices.MR3K4_KBO_VFS_Interface.q_xPRESS_OK_IG3 <-> FSVTask Inputs/GVL_FS_Devices.MR3K4_KBO_VFS_1.i_xPress_OK_IG3
//     PlcTask Outputs/GVL_FS_Devices.MR4K4_KBO_VFS_Interface.q_xPRESS_OK_IG1 <-> FSVTask Inputs/GVL_FS_Devices.MR4K4_KBO_VFS_1.i_xPress_OK_IG1
//     PlcTask Outputs/GVL_FS_Devices.MR4K4_KBO_VFS_Interface.q_xPRESS_OK_IG2 <-> FSVTask Inputs/GVL_FS_Devices.MR4K4_KBO_VFS_1.i_xPress_OK_IG2
//     PlcTask Outputs/GVL_FS_Devices.MR4K4_KBO_VFS_Interface.q_xPRESS_OK_IG3 <-> FSVTask Inputs/GVL_FS_Devices.MR4K4_KBO_VFS_1.i_xPress_OK_IG3
//     PlcTask Outputs/GVL_FS_Devices.MR3K4_KBO_VFS_Interface.q_xVAC_FAULT_Reset <-> FSVTask Inputs/GVL_FS_Devices.MR3K4_KBO_VFS_1.i_xVAC_FAULT_Reset
//     PlcTask Outputs/GVL_FS_Devices.MR4K4_KBO_VFS_Interface.q_xVAC_FAULT_Reset <-> FSVTask Inputs/GVL_FS_Devices.MR4K4_KBO_VFS_1.i_xVAC_FAULT_Reset
//     PlcTask Outputs/GVL_FS_Devices.MR3K4_KBO_VFS_Interface.q_xVetoValveClosed <-> FSVTask Inputs/GVL_FS_Devices.MR3K4_KBO_VFS_1.i_xVetoValveClosed
//     PlcTask Outputs/GVL_FS_Devices.MR4K4_KBO_VFS_Interface.q_xVetoValveClosed <-> FSVTask Inputs/GVL_FS_Devices.MR4K4_KBO_VFS_1.i_xVetoValveClosed
//     PlcTask Outputs/GVL_FS_Devices.MR3K4_KBO_VFS_Interface.q_xVetoValveOpenDO <-> FSVTask Inputs/GVL_FS_Devices.MR3K4_KBO_VFS_1.i_xVetoValveOpenDO
//     PlcTask Outputs/GVL_FS_Devices.MR4K4_KBO_VFS_Interface.q_xVetoValveOpenDO <-> FSVTask Inputs/GVL_FS_Devices.MR4K4_KBO_VFS_1.i_xVetoValveOpenDO
//     PlcTask Outputs/GVL_FS_Devices.TV1K4_VFS_Interface.q_ResetFaultCounter <-> FSVTask Inputs/GVL_FS_Devices.TV1K4_VFS_1.i_ResetFaultCounter
//     PlcTask Outputs/GVL_FS_Devices.TV1K4_VFS_Interface.q_e2OO3_MODE <-> FSVTask Inputs/GVL_FS_Devices.TV1K4_VFS_1.i_e2OO3_MODE
//     PlcTask Outputs/GVL_FS_Devices.TV1K4_VFS_Interface.q_xCLS_SW <-> FSVTask Inputs/GVL_FS_Devices.TV1K4_VFS_1.i_xCLS_SW
//     PlcTask Outputs/GVL_FS_Devices.TV1K4_VFS_Interface.q_xOPN_SW <-> FSVTask Inputs/GVL_FS_Devices.TV1K4_VFS_1.i_xOPN_SW
//     PlcTask Outputs/GVL_FS_Devices.TV1K4_VFS_Interface.q_xOverrideMode <-> FSVTask Inputs/GVL_FS_Devices.TV1K4_VFS_1.i_xOverrideMode
//     PlcTask Outputs/GVL_FS_Devices.TV1K4_VFS_Interface.q_xOverrideOpen <-> FSVTask Inputs/GVL_FS_Devices.TV1K4_VFS_1.i_xOverrideOpen
//     PlcTask Outputs/GVL_FS_Devices.TV1K4_VFS_Interface.q_xPRESS_OK_IG1 <-> FSVTask Inputs/GVL_FS_Devices.TV1K4_VFS_1.i_xPress_OK_IG1
//     PlcTask Outputs/GVL_FS_Devices.TV1K4_VFS_Interface.q_xPRESS_OK_IG2 <-> FSVTask Inputs/GVL_FS_Devices.TV1K4_VFS_1.i_xPress_OK_IG2
//     PlcTask Outputs/GVL_FS_Devices.TV1K4_VFS_Interface.q_xPRESS_OK_IG3 <-> FSVTask Inputs/GVL_FS_Devices.TV1K4_VFS_1.i_xPress_OK_IG3
//     PlcTask Outputs/GVL_FS_Devices.TV1K4_VFS_Interface.q_xVAC_FAULT_Reset <-> FSVTask Inputs/GVL_FS_Devices.TV1K4_VFS_1.i_xVAC_FAULT_Reset
//     PlcTask Outputs/GVL_FS_Devices.TV1K4_VFS_Interface.q_xVetoValveClosed <-> FSVTask Inputs/GVL_FS_Devices.TV1K4_VFS_1.i_xVetoValveClosed
//     PlcTask Outputs/GVL_FS_Devices.TV1K4_VFS_Interface.q_xVetoValveOpenDO <-> FSVTask Inputs/GVL_FS_Devices.TV1K4_VFS_1.i_xVetoValveOpenDO

CONFIGURATION PLC_TMO_VAC
    RESOURCE PLC ON TwinCAT3
        TASK ComTask(INTERVAL := T#11ms, PRIORITY := 30);
        TASK FSVTask(INTERVAL := T#2ms, PRIORITY := 15);
        TASK PlcTask(INTERVAL := T#10ms, PRIORITY := 20);
        PROGRAM PRG_COM WITH ComTask : PRG_COM;
        PROGRAM PRG_FSV WITH FSVTask : PRG_FSV;
        PROGRAM MAIN WITH PlcTask : MAIN;
    END_RESOURCE
END_CONFIGURATION

// ---- DUTs/E_STATES.TcDUT
{attribute 'qualified_only'}
{attribute 'strict'}
TYPE E_STATES :
(
    INIT := 0,
    SETUP,
    OVERRIDE,
    READY,
    NOT_SAFE
);
END_TYPE

// ---- GVLs/GVL_COM.TcGVL
VAR_GLOBAL
    // Define COM Ports/Buffers incl. library Tc2_SerialCom

    //PA1K4_IP1_PTM_01 , 02 and 03
    //K4S2_02_E10
    K4S2_02_E10_SerialRXBuffer : ComBuffer;
    K4S2_02_E10_SerialTXBuffer : ComBuffer;

    // Serial Terminal
    K4S2_02_E10_fbSerialLineControl: SerialLineControl;

    //SERIAL IO //K4S2_02_E10 (EL6021)
    {attribute	'TcLinkTo'	:=	'.Status:=TIIB[K4S2_02_E10 (EL6021)]^COM TxPDO-Map Inputs^Status;
                                 .D[0]:=TIIB[K4S2_02_E10 (EL6021)]^COM TxPDO-Map Inputs^Data In 0;
                                 .D[1]:=TIIB[K4S2_02_E10 (EL6021)]^COM TxPDO-Map Inputs^Data In 1;
                                 .D[2]:=TIIB[K4S2_02_E10 (EL6021)]^COM TxPDO-Map Inputs^Data In 2;
                                 .D[3]:=TIIB[K4S2_02_E10 (EL6021)]^COM TxPDO-Map Inputs^Data In 3;
                                 .D[4]:=TIIB[K4S2_02_E10 (EL6021)]^COM TxPDO-Map Inputs^Data In 4;
                                 .D[5]:=TIIB[K4S2_02_E10 (EL6021)]^COM TxPDO-Map Inputs^Data In 5;
                                 .D[6]:=TIIB[K4S2_02_E10 (EL6021)]^COM TxPDO-Map Inputs^Data In 6;
                                 .D[7]:=TIIB[K4S2_02_E10 (EL6021)]^COM TxPDO-Map Inputs^Data In 7;
                                 .D[8]:=TIIB[K4S2_02_E10 (EL6021)]^COM TxPDO-Map Inputs^Data In 8;
                                 .D[9]:=TIIB[K4S2_02_E10 (EL6021)]^COM TxPDO-Map Inputs^Data In 9;
                                 .D[10]:=TIIB[K4S2_02_E10 (EL6021)]^COM TxPDO-Map Inputs^Data In 10;
                                 .D[11]:=TIIB[K4S2_02_E10 (EL6021)]^COM TxPDO-Map Inputs^Data In 11;
                                 .D[12]:=TIIB[K4S2_02_E10 (EL6021)]^COM TxPDO-Map Inputs^Data In 12;
                                 .D[13]:=TIIB[K4S2_02_E10 (EL6021)]^COM TxPDO-Map Inputs^Data In 13;
                                 .D[14]:=TIIB[K4S2_02_E10 (EL6021)]^COM TxPDO-Map Inputs^Data In 14;
                                 .D[15]:=TIIB[K4S2_02_E10 (EL6021)]^COM TxPDO-Map Inputs^Data In 15;
                                 .D[16]:=TIIB[K4S2_02_E10 (EL6021)]^COM TxPDO-Map Inputs^Data In 16;
                                 .D[17]:=TIIB[K4S2_02_E10 (EL6021)]^COM TxPDO-Map Inputs^Data In 17;
                                 .D[18]:=TIIB[K4S2_02_E10 (EL6021)]^COM TxPDO-Map Inputs^Data In 18;
                                 .D[19]:=TIIB[K4S2_02_E10 (EL6021)]^COM TxPDO-Map Inputs^Data In 19;
                                 .D[20]:=TIIB[K4S2_02_E10 (EL6021)]^COM TxPDO-Map Inputs^Data In 20;
                                 .D[21]:=TIIB[K4S2_02_E10 (EL6021)]^COM TxPDO-Map Inputs^Data In 21
    '}
    K4S2_02_E10_stComIn		AT %I*	:	EL6inData22B;
    {attribute	'TcLinkTo'	:=	'.Ctrl:=TIIB[K4S2_02_E10 (EL6021)]^COM RxPDO-Map Outputs^Ctrl;
                                 .D[0]:=TIIB[K4S2_02_E10 (EL6021)]^COM RxPDO-Map Outputs^Data Out 0;
                                 .D[1]:=TIIB[K4S2_02_E10 (EL6021)]^COM RxPDO-Map Outputs^Data Out 1;
                                 .D[2]:=TIIB[K4S2_02_E10 (EL6021)]^COM RxPDO-Map Outputs^Data Out 2;
                                 .D[3]:=TIIB[K4S2_02_E10 (EL6021)]^COM RxPDO-Map Outputs^Data Out 3;
                                 .D[4]:=TIIB[K4S2_02_E10 (EL6021)]^COM RxPDO-Map Outputs^Data Out 4;
                                 .D[5]:=TIIB[K4S2_02_E10 (EL6021)]^COM RxPDO-Map Outputs^Data Out 5;
                                 .D[6]:=TIIB[K4S2_02_E10 (EL6021)]^COM RxPDO-Map Outputs^Data Out 6;
                                 .D[7]:=TIIB[K4S2_02_E10 (EL6021)]^COM RxPDO-Map Outputs^Data Out 7;
                                 .D[8]:=TIIB[K4S2_02_E10 (EL6021)]^COM RxPDO-Map Outputs^Data Out 8;
                                 .D[9]:=TIIB[K4S2_02_E10 (EL6021)]^COM RxPDO-Map Outputs^Data Out 9;
                                 .D[10]:=TIIB[K4S2_02_E10 (EL6021)]^COM RxPDO-Map Outputs^Data Out 10;
                                 .D[11]:=TIIB[K4S2_02_E10 (EL6021)]^COM RxPDO-Map Outputs^Data Out 11;
                                 .D[12]:=TIIB[K4S2_02_E10 (EL6021)]^COM RxPDO-Map Outputs^Data Out 12;
                                 .D[13]:=TIIB[K4S2_02_E10 (EL6021)]^COM RxPDO-Map Outputs^Data Out 13;
                                 .D[14]:=TIIB[K4S2_02_E10 (EL6021)]^COM RxPDO-Map Outputs^Data Out 14;
                                 .D[15]:=TIIB[K4S2_02_E10 (EL6021)]^COM RxPDO-Map Outputs^Data Out 15;
                                 .D[16]:=TIIB[K4S2_02_E10 (EL6021)]^COM RxPDO-Map Outputs^Data Out 16;
                                 .D[17]:=TIIB[K4S2_02_E10 (EL6021)]^COM RxPDO-Map Outputs^Data Out 17;
                                 .D[18]:=TIIB[K4S2_02_E10 (EL6021)]^COM RxPDO-Map Outputs^Data Out 18;
                                 .D[19]:=TIIB[K4S2_02_E10 (EL6021)]^COM RxPDO-Map Outputs^Data Out 19;
                                 .D[20]:=TIIB[K4S2_02_E10 (EL6021)]^COM RxPDO-Map Outputs^Data Out 20;
                                 .D[21]:=TIIB[K4S2_02_E10 (EL6021)]^COM RxPDO-Map Outputs^Data Out 21
    '}
    K4S2_02_E10_stComOut		AT %Q*	:	EL6outData22B;


    //Granite 2
    //LI3K4_IP1_OUT_PTM_01-TM1K4_PTM_01-IM5K4_PPM_PTM_01
    //K4S6_01_E5 (EL6021)
    K4S6_01_E5_SerialRXBuffer : ComBuffer;
    K4S6_01_E5_SerialTXBuffer : ComBuffer;

    // Serial Terminal
    K4S6_01_E5_fbSerialLineControl: SerialLineControl;

    //Serial IO
        {attribute	'TcLinkTo'	:=	'.Status:=TIIB[K4S6_01_E5 (EL6021)]^COM TxPDO-Map Inputs^Status;
                                 .D[0]:=TIIB[K4S6_01_E5 (EL6021)]^COM TxPDO-Map Inputs^Data In 0;
                                 .D[1]:=TIIB[K4S6_01_E5 (EL6021)]^COM TxPDO-Map Inputs^Data In 1;
                                 .D[2]:=TIIB[K4S6_01_E5 (EL6021)]^COM TxPDO-Map Inputs^Data In 2;
                                 .D[3]:=TIIB[K4S6_01_E5 (EL6021)]^COM TxPDO-Map Inputs^Data In 3;
                                 .D[4]:=TIIB[K4S6_01_E5 (EL6021)]^COM TxPDO-Map Inputs^Data In 4;
                                 .D[5]:=TIIB[K4S6_01_E5 (EL6021)]^COM TxPDO-Map Inputs^Data In 5;
                                 .D[6]:=TIIB[K4S6_01_E5 (EL6021)]^COM TxPDO-Map Inputs^Data In 6;
                                 .D[7]:=TIIB[K4S6_01_E5 (EL6021)]^COM TxPDO-Map Inputs^Data In 7;
                                 .D[8]:=TIIB[K4S6_01_E5 (EL6021)]^COM TxPDO-Map Inputs^Data In 8;
                                 .D[9]:=TIIB[K4S6_01_E5 (EL6021)]^COM TxPDO-Map Inputs^Data In 9;
                                 .D[10]:=TIIB[K4S6_01_E5 (EL6021)]^COM TxPDO-Map Inputs^Data In 10;
                                 .D[11]:=TIIB[K4S6_01_E5 (EL6021)]^COM TxPDO-Map Inputs^Data In 11;
                                 .D[12]:=TIIB[K4S6_01_E5 (EL6021)]^COM TxPDO-Map Inputs^Data In 12;
                                 .D[13]:=TIIB[K4S6_01_E5 (EL6021)]^COM TxPDO-Map Inputs^Data In 13;
                                 .D[14]:=TIIB[K4S6_01_E5 (EL6021)]^COM TxPDO-Map Inputs^Data In 14;
                                 .D[15]:=TIIB[K4S6_01_E5 (EL6021)]^COM TxPDO-Map Inputs^Data In 15;
                                 .D[16]:=TIIB[K4S6_01_E5 (EL6021)]^COM TxPDO-Map Inputs^Data In 16;
                                 .D[17]:=TIIB[K4S6_01_E5 (EL6021)]^COM TxPDO-Map Inputs^Data In 17;
                                 .D[18]:=TIIB[K4S6_01_E5 (EL6021)]^COM TxPDO-Map Inputs^Data In 18;
                                 .D[19]:=TIIB[K4S6_01_E5 (EL6021)]^COM TxPDO-Map Inputs^Data In 19;
                                 .D[20]:=TIIB[K4S6_01_E5 (EL6021)]^COM TxPDO-Map Inputs^Data In 20;
                                 .D[21]:=TIIB[K4S6_01_E5 (EL6021)]^COM TxPDO-Map Inputs^Data In 21
    '}
    K4S6_01_E5_stComIn		AT %I*	:	EL6inData22B;
    {attribute	'TcLinkTo'	:=	'.Ctrl:=TIIB[K4S6_01_E5 (EL6021)]^COM RxPDO-Map Outputs^Ctrl;
                                 .D[0]:=TIIB[K4S6_01_E5 (EL6021)]^COM RxPDO-Map Outputs^Data Out 0;
                                 .D[1]:=TIIB[K4S6_01_E5 (EL6021)]^COM RxPDO-Map Outputs^Data Out 1;
                                 .D[2]:=TIIB[K4S6_01_E5 (EL6021)]^COM RxPDO-Map Outputs^Data Out 2;
                                 .D[3]:=TIIB[K4S6_01_E5 (EL6021)]^COM RxPDO-Map Outputs^Data Out 3;
                                 .D[4]:=TIIB[K4S6_01_E5 (EL6021)]^COM RxPDO-Map Outputs^Data Out 4;
                                 .D[5]:=TIIB[K4S6_01_E5 (EL6021)]^COM RxPDO-Map Outputs^Data Out 5;
                                 .D[6]:=TIIB[K4S6_01_E5 (EL6021)]^COM RxPDO-Map Outputs^Data Out 6;
                                 .D[7]:=TIIB[K4S6_01_E5 (EL6021)]^COM RxPDO-Map Outputs^Data Out 7;
                                 .D[8]:=TIIB[K4S6_01_E5 (EL6021)]^COM RxPDO-Map Outputs^Data Out 8;
                                 .D[9]:=TIIB[K4S6_01_E5 (EL6021)]^COM RxPDO-Map Outputs^Data Out 9;
                                 .D[10]:=TIIB[K4S6_01_E5 (EL6021)]^COM RxPDO-Map Outputs^Data Out 10;
                                 .D[11]:=TIIB[K4S6_01_E5 (EL6021)]^COM RxPDO-Map Outputs^Data Out 11;
                                 .D[12]:=TIIB[K4S6_01_E5 (EL6021)]^COM RxPDO-Map Outputs^Data Out 12;
                                 .D[13]:=TIIB[K4S6_01_E5 (EL6021)]^COM RxPDO-Map Outputs^Data Out 13;
                                 .D[14]:=TIIB[K4S6_01_E5 (EL6021)]^COM RxPDO-Map Outputs^Data Out 14;
                                 .D[15]:=TIIB[K4S6_01_E5 (EL6021)]^COM RxPDO-Map Outputs^Data Out 15;
                                 .D[16]:=TIIB[K4S6_01_E5 (EL6021)]^COM RxPDO-Map Outputs^Data Out 16;
                                 .D[17]:=TIIB[K4S6_01_E5 (EL6021)]^COM RxPDO-Map Outputs^Data Out 17;
                                 .D[18]:=TIIB[K4S6_01_E5 (EL6021)]^COM RxPDO-Map Outputs^Data Out 18;
                                 .D[19]:=TIIB[K4S6_01_E5 (EL6021)]^COM RxPDO-Map Outputs^Data Out 19;
                                 .D[20]:=TIIB[K4S6_01_E5 (EL6021)]^COM RxPDO-Map Outputs^Data Out 20;
                                 .D[21]:=TIIB[K4S6_01_E5 (EL6021)]^COM RxPDO-Map Outputs^Data Out 21
    '}
    K4S6_01_E5_stComOut		AT %Q*	:	EL6outData22B;

    //IM4K4_PPM_PTM_01
    //K4S2_02_E17 (EL6001)
    K4S2_02_E17_SerialRXBuffer : ComBuffer;
    K4S2_02_E17_SerialTXBuffer : ComBuffer;

    // Serial Terminal
    K4S2_02_E17_fbSerialLineControl: SerialLineControl;
        //Serial IO
        {attribute	'TcLinkTo'	:=	'.Status:=TIIB[K4S2_02_E17 (EL6001)]^COM Inputs^Status;
                                 .D[0]:=TIIB[K4S2_02_E17 (EL6001)]^COM Inputs^Data In 0;
                                 .D[1]:=TIIB[K4S2_02_E17 (EL6001)]^COM Inputs^Data In 1;
                                 .D[2]:=TIIB[K4S2_02_E17 (EL6001)]^COM Inputs^Data In 2;
                                 .D[3]:=TIIB[K4S2_02_E17 (EL6001)]^COM Inputs^Data In 3;
                                 .D[4]:=TIIB[K4S2_02_E17 (EL6001)]^COM Inputs^Data In 4;
                                 .D[5]:=TIIB[K4S2_02_E17 (EL6001)]^COM Inputs^Data In 5;
                                 .D[6]:=TIIB[K4S2_02_E17 (EL6001)]^COM Inputs^Data In 6;
                                 .D[7]:=TIIB[K4S2_02_E17 (EL6001)]^COM Inputs^Data In 7;
                                 .D[8]:=TIIB[K4S2_02_E17 (EL6001)]^COM Inputs^Data In 8;
                                 .D[9]:=TIIB[K4S2_02_E17 (EL6001)]^COM Inputs^Data In 9;
                                 .D[10]:=TIIB[K4S2_02_E17 (EL6001)]^COM Inputs^Data In 10;
                                 .D[11]:=TIIB[K4S2_02_E17 (EL6001)]^COM Inputs^Data In 11;
                                 .D[12]:=TIIB[K4S2_02_E17 (EL6001)]^COM Inputs^Data In 12;
                                 .D[13]:=TIIB[K4S2_02_E17 (EL6001)]^COM Inputs^Data In 13;
                                 .D[14]:=TIIB[K4S2_02_E17 (EL6001)]^COM Inputs^Data In 14;
                                 .D[15]:=TIIB[K4S2_02_E17 (EL6001)]^COM Inputs^Data In 15;
                                 .D[16]:=TIIB[K4S2_02_E17 (EL6001)]^COM Inputs^Data In 16;
                                 .D[17]:=TIIB[K4S2_02_E17 (EL6001)]^COM Inputs^Data In 17;
                                 .D[18]:=TIIB[K4S2_02_E17 (EL6001)]^COM Inputs^Data In 18;
                                 .D[19]:=TIIB[K4S2_02_E17 (EL6001)]^COM Inputs^Data In 19;
                                 .D[20]:=TIIB[K4S2_02_E17 (EL6001)]^COM Inputs^Data In 20;
                                 .D[21]:=TIIB[K4S2_02_E17 (EL6001)]^COM Inputs^Data In 21
    '}
    K4S2_02_E17_stComIn		AT %I*	:	EL6inData22B;
    {attribute	'TcLinkTo'	:=	'.Ctrl:=TIIB[K4S2_02_E17 (EL6001)]^COM Outputs^Ctrl;
                                 .D[0]:=TIIB[K4S2_02_E17 (EL6001)]^COM Outputs^Data Out 0;
                                 .D[1]:=TIIB[K4S2_02_E17 (EL6001)]^COM Outputs^Data Out 1;
                                 .D[2]:=TIIB[K4S2_02_E17 (EL6001)]^COM Outputs^Data Out 2;
                                 .D[3]:=TIIB[K4S2_02_E17 (EL6001)]^COM Outputs^Data Out 3;
                                 .D[4]:=TIIB[K4S2_02_E17 (EL6001)]^COM Outputs^Data Out 4;
                                 .D[5]:=TIIB[K4S2_02_E17 (EL6001)]^COM Outputs^Data Out 5;
                                 .D[6]:=TIIB[K4S2_02_E17 (EL6001)]^COM Outputs^Data Out 6;
                                 .D[7]:=TIIB[K4S2_02_E17 (EL6001)]^COM Outputs^Data Out 7;
                                 .D[8]:=TIIB[K4S2_02_E17 (EL6001)]^COM Outputs^Data Out 8;
                                 .D[9]:=TIIB[K4S2_02_E17 (EL6001)]^COM Outputs^Data Out 9;
                                 .D[10]:=TIIB[K4S2_02_E17 (EL6001)]^COM Outputs^Data Out 10;
                                 .D[11]:=TIIB[K4S2_02_E17 (EL6001)]^COM Outputs^Data Out 11;
                                 .D[12]:=TIIB[K4S2_02_E17 (EL6001)]^COM Outputs^Data Out 12;
                                 .D[13]:=TIIB[K4S2_02_E17 (EL6001)]^COM Outputs^Data Out 13;
                                 .D[14]:=TIIB[K4S2_02_E17 (EL6001)]^COM Outputs^Data Out 14;
                                 .D[15]:=TIIB[K4S2_02_E17 (EL6001)]^COM Outputs^Data Out 15;
                                 .D[16]:=TIIB[K4S2_02_E17 (EL6001)]^COM Outputs^Data Out 16;
                                 .D[17]:=TIIB[K4S2_02_E17 (EL6001)]^COM Outputs^Data Out 17;
                                 .D[18]:=TIIB[K4S2_02_E17 (EL6001)]^COM Outputs^Data Out 18;
                                 .D[19]:=TIIB[K4S2_02_E17 (EL6001)]^COM Outputs^Data Out 19;
                                 .D[20]:=TIIB[K4S2_02_E17 (EL6001)]^COM Outputs^Data Out 20;
                                 .D[21]:=TIIB[K4S2_02_E17 (EL6001)]^COM Outputs^Data Out 21
    '}
    K4S2_02_E17_stComOut		AT %Q*	:	EL6outData22B;

    //LI1K4_IP1_PTM_01
    //K4S2_02_E18 (EL6001)

    // Define COM Ports/Buffers incl. library Tc2_SerialCom
    K4S2_02_E18_SerialRXBuffer : ComBuffer;
    K4S2_02_E18_SerialTXBuffer : ComBuffer;

    // Serial Terminal
    K4S2_02_E18_fbSerialLineControl: SerialLineControl;

    //SERIAL IO
    {attribute	'TcLinkTo'	:=	'.Status:=TIIB[K4S2_02_E18 (EL6001)]^COM Inputs^Status;
                                 .D[0]:=TIIB[K4S2_02_E18 (EL6001)]^COM Inputs^Data In 0;
                                 .D[1]:=TIIB[K4S2_02_E18 (EL6001)]^COM Inputs^Data In 1;
                                 .D[2]:=TIIB[K4S2_02_E18 (EL6001)]^COM Inputs^Data In 2;
                                 .D[3]:=TIIB[K4S2_02_E18 (EL6001)]^COM Inputs^Data In 3;
                                 .D[4]:=TIIB[K4S2_02_E18 (EL6001)]^COM Inputs^Data In 4;
                                 .D[5]:=TIIB[K4S2_02_E18 (EL6001)]^COM Inputs^Data In 5;
                                 .D[6]:=TIIB[K4S2_02_E18 (EL6001)]^COM Inputs^Data In 6;
                                 .D[7]:=TIIB[K4S2_02_E18 (EL6001)]^COM Inputs^Data In 7;
                                 .D[8]:=TIIB[K4S2_02_E18 (EL6001)]^COM Inputs^Data In 8;
                                 .D[9]:=TIIB[K4S2_02_E18 (EL6001)]^COM Inputs^Data In 9;
                                 .D[10]:=TIIB[K4S2_02_E18 (EL6001)]^COM Inputs^Data In 10;
                                 .D[11]:=TIIB[K4S2_02_E18 (EL6001)]^COM Inputs^Data In 11;
                                 .D[12]:=TIIB[K4S2_02_E18 (EL6001)]^COM Inputs^Data In 12;
                                 .D[13]:=TIIB[K4S2_02_E18 (EL6001)]^COM Inputs^Data In 13;
                                 .D[14]:=TIIB[K4S2_02_E18 (EL6001)]^COM Inputs^Data In 14;
                                 .D[15]:=TIIB[K4S2_02_E18 (EL6001)]^COM Inputs^Data In 15;
                                 .D[16]:=TIIB[K4S2_02_E18 (EL6001)]^COM Inputs^Data In 16;
                                 .D[17]:=TIIB[K4S2_02_E18 (EL6001)]^COM Inputs^Data In 17;
                                 .D[18]:=TIIB[K4S2_02_E18 (EL6001)]^COM Inputs^Data In 18;
                                 .D[19]:=TIIB[K4S2_02_E18 (EL6001)]^COM Inputs^Data In 19;
                                 .D[20]:=TIIB[K4S2_02_E18 (EL6001)]^COM Inputs^Data In 20;
                                 .D[21]:=TIIB[K4S2_02_E18 (EL6001)]^COM Inputs^Data In 21
    '}
    K4S2_02_E18_stComIn		AT %I*	:	EL6inData22B;
    {attribute	'TcLinkTo'	:=	'.Ctrl:=TIIB[K4S2_02_E18 (EL6001)]^COM Outputs^Ctrl;
                                 .D[0]:=TIIB[K4S2_02_E18 (EL6001)]^COM Outputs^Data Out 0;
                                 .D[1]:=TIIB[K4S2_02_E18 (EL6001)]^COM Outputs^Data Out 1;
                                 .D[2]:=TIIB[K4S2_02_E18 (EL6001)]^COM Outputs^Data Out 2;
                                 .D[3]:=TIIB[K4S2_02_E18 (EL6001)]^COM Outputs^Data Out 3;
                                 .D[4]:=TIIB[K4S2_02_E18 (EL6001)]^COM Outputs^Data Out 4;
                                 .D[5]:=TIIB[K4S2_02_E18 (EL6001)]^COM Outputs^Data Out 5;
                                 .D[6]:=TIIB[K4S2_02_E18 (EL6001)]^COM Outputs^Data Out 6;
                                 .D[7]:=TIIB[K4S2_02_E18 (EL6001)]^COM Outputs^Data Out 7;
                                 .D[8]:=TIIB[K4S2_02_E18 (EL6001)]^COM Outputs^Data Out 8;
                                 .D[9]:=TIIB[K4S2_02_E18 (EL6001)]^COM Outputs^Data Out 9;
                                 .D[10]:=TIIB[K4S2_02_E18 (EL6001)]^COM Outputs^Data Out 10;
                                 .D[11]:=TIIB[K4S2_02_E18 (EL6001)]^COM Outputs^Data Out 11;
                                 .D[12]:=TIIB[K4S2_02_E18 (EL6001)]^COM Outputs^Data Out 12;
                                 .D[13]:=TIIB[K4S2_02_E18 (EL6001)]^COM Outputs^Data Out 13;
                                 .D[14]:=TIIB[K4S2_02_E18 (EL6001)]^COM Outputs^Data Out 14;
                                 .D[15]:=TIIB[K4S2_02_E18 (EL6001)]^COM Outputs^Data Out 15;
                                 .D[16]:=TIIB[K4S2_02_E18 (EL6001)]^COM Outputs^Data Out 16;
                                 .D[17]:=TIIB[K4S2_02_E18 (EL6001)]^COM Outputs^Data Out 17;
                                 .D[18]:=TIIB[K4S2_02_E18 (EL6001)]^COM Outputs^Data Out 18;
                                 .D[19]:=TIIB[K4S2_02_E18 (EL6001)]^COM Outputs^Data Out 19;
                                 .D[20]:=TIIB[K4S2_02_E18 (EL6001)]^COM Outputs^Data Out 20;
                                 .D[21]:=TIIB[K4S2_02_E18 (EL6001)]^COM Outputs^Data Out 21
    '}
    K4S2_02_E18_stComOut		AT %Q*	:	EL6outData22B;



END_VAR

// ---- GVLs/GVL_DREAM_ECAT.TcGVL
//{attribute 'qualified_only'}
VAR_GLOBAL
   (* These variables are for DREAM EtherCat bridge *)
   (*ETHERCAT BRIDGE COM STATUS*)
   //EL6695 TxPDO state
   //0: Other side is in OP state, >0: Error
   {attribute 'TcLinkTo' := 'TIIB[CX0_E13 (EK1122)]^DREAM_ECAT^SYNC Inputs^TxPDO state'}
   bDreamEcatBridge_TxPDO_state AT %I* : BOOL;

   //0: External device connected, 1: External device not connected
   {attribute 'TcLinkTo' := 'TIIB[CX0_E13 (EK1122)]^DREAM_ECAT^SYNC Inputs^External device not connected'}
   bDreamEcatBridge_External_device_not_connected AT %I* : BOOL;

   //0 = Data valid, 1 = Data invalid
   {attribute 'TcLinkTo' := 'TIIB[CX0_E13 (EK1122)]^DREAM_ECAT^WcState^WcState'}
   bDreamEcatBridge_WcState AT %I* : BOOL;

   //Detecting ethercat communication errror
   {attribute 'pytmc' := 'pv: TMO:DREAM:ENDSTATION:ETHERCAT_ERROR'}
   bDREAM_ECAT_COM_ERROR : BOOL;

   //DREAM EL6695 OUTPUTS
   {attribute 'TcLinkTo' := 	'TIIB[CX0_E13 (EK1122)]^DREAM_ECAT^IO Outputs^HUTCH_PLC_NAME'}
   sHutchPlcName	AT %Q*	: STRING(8) := 'TMO';

   //DREAM EL6695 INPUTS
   {attribute 'pytmc'    := 'pv: TMO:IP2:PLC:NAME'}
   {attribute 'TcLinkTo' := 'TIIB[CX0_E13 (EK1122)]^DREAM_ECAT^IO Inputs^ENDSTATION_PLC_NAME'}
   DREAM_PLC_NAME AT %I*  : STRING(8);

   {attribute 'pytmc'    := 'pv: TMO:DREAM:TURBOS:ALL_AT_SPD'}
   {attribute 'TcLinkTo' := 'TIIB[CX0_E13 (EK1122)]^DREAM_ECAT^IO Inputs^DREAM_TURBOS_ALL_AtSpd'}
   DREAM_TURBOS_ALL_AtSpd AT %I* : BOOL;

   {attribute 'pytmc'    := 'pv: TMO:DREAM:HV_SAFETY_ENABLE'}
   {attribute 'TcLinkTo' := 'TIIB[CX0_E13 (EK1122)]^DREAM_ECAT^IO Inputs^DREAM_HV_SAFETY_ENABLE'}
   DREAM_HV_SAFETY_ENABLE AT %I* : BOOL;

   {attribute 'pytmc' :=' pv: TMO:DREAM:MAIN:GAUGE'}
   {attribute 'TcLinkTo' := '.i_xAT_VAC             := TIIB[CX0_E13 (EK1122)]^DREAM_ECAT^IO Inputs^DREAM_MAIN_xAT_VAC;
                             .i_xPRESS_OK           := TIIB[CX0_E13 (EK1122)]^DREAM_ECAT^IO Inputs^DREAM_MAIN_xPRESS_OK;
                             .i_rPRESS              := TIIB[CX0_E13 (EK1122)]^DREAM_ECAT^IO Inputs^DREAM_MAIN_rPRESS
   '}
   DREAM_MAIN_GAUGE : FB_Gauge_Interface;

   //gauge structure, which can be override if there is an Ethercat communication error
   stDreamMainGauge : ST_VG;

   //Window valve interface
   {attribute 'TcLinkTo' := 	'TIIB[CX0_E13 (EK1122)]^DREAM_ECAT^IO Outputs^TMO_MR5K4_VWC_CLOSED_LS'}
   bTMO_MR5K4_VWC_CLOSED_LS	AT %Q*	: BOOL;

   {attribute 'TcLinkTo' := 	'TIIB[CX0_E13 (EK1122)]^DREAM_ECAT^IO Outputs^TMO_TM2K4_VWC_CLOSED_LS'}
   bTMO_TM2K4_VWC_CLOSED_LS	AT %Q*	: BOOL;

   {attribute 'TcLinkTo' := 	'TIIB[CX0_E13 (EK1122)]^DREAM_ECAT^IO Outputs^TMO_MR5K4_VWC_OPEN_LS'}
   bTMO_MR5K4_VWC_OPEN_LS	AT %Q*	: BOOL;

   {attribute 'TcLinkTo' := 	'TIIB[CX0_E13 (EK1122)]^DREAM_ECAT^IO Outputs^TMO_TM2K4_VWC_OPEN_LS'}
   bTMO_TM2K4_VWC_OPEN_LS	AT %Q*	: BOOL;

   {attribute 'TcLinkTo' := 'TIIB[CX0_E13 (EK1122)]^DREAM_ECAT^IO Inputs^CLOSE_TMO_MR5K4_VWC'}
   bCLOSE_TMO_MR5K4_VWC AT %I* : BOOL;

   {attribute 'TcLinkTo' := 'TIIB[CX0_E13 (EK1122)]^DREAM_ECAT^IO Inputs^CLOSE_TMO_TM2K4_VWC '}
   bCLOSE_TMO_TM2K4_VWC  AT %I* : BOOL;
END_VAR

// ---- GVLs/GVL_FEE_Device.TcGVL
//{attribute 'qualified_only'}
VAR_GLOBAL

(* upstream vacuum ok *)
   {attribute 'pytmc' :=' pv: USVAC:OK:HI '}
   {attribute 'TcLinkTo' := 	' := 	TIIB[CX0_E2_EXILK (EL1008)]^Channel 1^Input	'}
   USVacOk_HI AT%I* : BOOL; (* upstream vacuum <10E-6, for mirror VGC interlock *)

     {attribute 'pytmc' :=' pv: USVAC:OK:LO '}
   {attribute 'TcLinkTo' := 	'	:= 	TIIB[CX0_E2_EXILK (EL1008)]^Channel 3^Input	'}
   USVacOk_LO AT%I* : BOOL; (* upstream vacuum <10E-4, for Ion pump interlock *)


(* Isolation gate valves*)

    {attribute 'pytmc' :=' pv: TV1K4:VGC:01 '}
    {attribute 'TcLinkTo' := 	'.i_xOpnLS	:=	TIIB[B940_K4S20_EB1  (EP2338-0002)]^Channel 1^Input;
                                 .i_xClsLS	:=	TIIB[B940_K4S20_EB1  (EP2338-0002)]^Channel 2^Input;
                                .q_xOPN_DO	:=	TIIB[B940_K4S20_EB1  (EP2338-0002)]^Channel 11^Output'}
    TV1K4_VGC_01: FB_VGC;

    {attribute 'pytmc' :=' pv: TV1K4:VGC:02 '}
    {attribute 'TcLinkTo' := 	'.i_xOpnLS	:=	TIIB[B940_K4S20_EB1  (EP2338-0002)]^Channel 5^Input;
                                 .i_xClsLS	:=	TIIB[B940_K4S20_EB1  (EP2338-0002)]^Channel 6^Input;
                                 .q_xOPN_DO	:=	TIIB[B940_K4S20_EB1  (EP2338-0002)]^Channel 15^Output'}
     TV1K4_VGC_02: FB_VGC;

    {attribute 'pytmc' :=' pv: ST3K4:PPS:VGC:01 '}
    {attribute 'TcLinkTo' := 	'.i_xOpnLS	:=	TIIB[B940_K4S33_EB1 (EP2338-0002)]^Channel 1^Input;
                                 .i_xClsLS	:=	TIIB[B940_K4S33_EB1 (EP2338-0002)]^Channel 2^Input;
                                 .q_xOPN_DO	:=	TIIB[B940_K4S33_EB1 (EP2338-0002)]^Channel 11^Output'}
    ST3K4_PPS_VGC_01 : FB_VGC;

(* Pirani & Cold Cathode*)



    {attribute 'pytmc' :=' pv: TV1K4:GPI:01 '}
    {attribute 'TcLinkTo' := 	'.i_iPRESS_R	:=	TIIB[B940_K4S20_EB2  (EP3174-0002)]^AI Standard Channel 1^Value	'}
    TV1K4_GPI_01 : FB_MKS275;


    {attribute 'pytmc' :=' pv: TV1K4:GCC:01 '}
    {attribute 'TcLinkTo' := 	'.i_iPRESS_R	:=	TIIB[B940_K4S20_EB2  (EP3174-0002)]^AI Standard Channel 2^Value;
                                 .q_xHV_DIS		:= 	TIIB[B940_K4S20_EB3 (EP2624-0002)]^Channel 1^Output	'}
    TV1K4_GCC_01 : FB_MKS500;

    {attribute 'pytmc' :=' pv: ST1K4:TEST:GPI:01 '}
    {attribute 'TcLinkTo' := 	'.i_iPRESS_R	:=	TIIB[B940_K4S24_EB1 (EP3174-0002)]^AI Standard Channel 1^Value		'}
    ST1K4_TEST_GPI_01 : FB_MKS275;


    {attribute 'pytmc' :=' pv: ST1K4:TEST:GCC:01 '}
    {attribute 'TcLinkTo' := 	'.i_iPRESS_R	:=	TIIB[B940_K4S24_EB1 (EP3174-0002)]^AI Standard Channel 2^Value;
                                 .q_xHV_DIS		:= 	TIIB[B940_K4S24_EB2 (EP2624-0002)]^Channel 1^Output	'}
    ST1K4_TEST_GCC_01 : FB_MKS500;


    {attribute 'pytmc' :=' pv: ST2K4:BCS:GPI:01 '}
    {attribute 'TcLinkTo' := 	'.i_iPRESS_R	:=	TIIB[B940_K4S28_EB1 (EP3174-0002)]^AI Standard Channel 1^Value	'}
    ST2K4_BCS_GPI_01 : FB_MKS275;

    {attribute 'pytmc' :=' pv: ST2K4:BCS:GCC:01 '}
    {attribute 'TcLinkTo' := 	'.i_iPRESS_R	:=	TIIB[B940_K4S28_EB1 (EP3174-0002)]^AI Standard Channel 2^Value;
                                 .q_xHV_DIS		:= 	TIIB[B940_K4S28_EB2 (EP2624-0002)]^Channel 1^Output	'}
    ST2K4_BCS_GCC_01 : FB_MKS500;


    {attribute 'pytmc' :=' pv: PC4K4:XTES:GPI:01 '}
    {attribute 'TcLinkTo' := 	'.i_iPRESS_R	:=	TIIB[B940_K4S33_EB2 (EP3174-0002)]^AI Standard Channel 1^Value	'}
    PC4K4_XTES_GPI_01 : FB_MKS275;

    {attribute 'pytmc' :=' pv: PC4K4:XTES:GCC:01 '}
    {attribute 'TcLinkTo' := 	'.i_iPRESS_R	:=	TIIB[B940_K4S33_EB2 (EP3174-0002)]^AI Standard Channel 2^Value;
                                 .q_xHV_DIS		:= 	TIIB[B940_K4S33_EB3 (EP2624-0002)]^Channel 1^Output	'}

    PC4K4_XTES_GCC_01 : FB_MKS500;

    {attribute 'pytmc' :=' pv: PC4K4:XTES:GCC:02 '}
    {attribute 'TcLinkTo' := 	'.i_iPRESS_R	:=	TIIB[B940_K4S33_EB2 (EP3174-0002)]^AI Standard Channel 3^Value;
                                 .q_xHV_DIS		:= 	TIIB[B940_K4S33_EB3 (EP2624-0002)]^Channel 2^Output'}
    PC4K4_XTES_GCC_02 : FB_MX7M;



(* Ion Pumps *)

    {attribute 'pytmc' :='
            pv: MR1K4:SOMS:PIP:01 '}
    {attribute 'TcLinkTo' := 	'.i_iPRESS		:=	TIIB[CX0_E6_QPC1 (EL3064)]^AI Standard Channel 1^Value;
                                 .i_xSP_DI		:= 	TIIB[CX0_E7_QPC1 (EL1004)]^Channel 1^Input;
                                 .q_xHVEna_DO	:= 	TIIB[CX0_E8_QPC1 (EL2794)]^Channel 1^Output
    '}
    MR1K4_SOMS_PIP_01 : FB_PIP_Gamma;

    {attribute 'pytmc' :=' pv: ST1K4:TEST:PIP:01 '}
    {attribute 'TcLinkTo' := 	'.i_iPRESS		:=	TIIB[CX0_E6_QPC1 (EL3064)]^AI Standard Channel 2^Value;
                                 .i_xSP_DI		:= 	TIIB[CX0_E7_QPC1 (EL1004)]^Channel 2^Input;
                                 .q_xHVEna_DO	:= 	TIIB[CX0_E8_QPC1 (EL2794)]^Channel 2^Output
    '}
    ST1K4_TEST_PIP_01 : FB_PIP_Gamma;

    {attribute 'pytmc' :=' pv: ST2K4:BCS:PIP:01 '}
    {attribute 'TcLinkTo' := 	'.i_iPRESS		:=	TIIB[CX0_E6_QPC1 (EL3064)]^AI Standard Channel 3^Value;
                                 .i_xSP_DI		:= 	TIIB[CX0_E7_QPC1 (EL1004)]^Channel 3^Input;
                                 .q_xHVEna_DO	:= 	TIIB[CX0_E8_QPC1 (EL2794)]^Channel 3^Output
    '}
    ST2K4_BCS_PIP_01 : FB_PIP_Gamma;

